# B&R Automation Studio project Snapshot
Automation Studio 4.9.2.46; technology packages: mapp 5.15.0, mappMotion 5.15.1

## Configuration Config1

CPU PC_any, AutomationRuntime D4.90, Build 4.1.2, Safety 0.0, Vc V4.72.2

### Task classes (Cpu.sw)
```
Cyclic#1 (cycle 10000 us):
  UserProgra <- UserProgram.prg
  TrakProgra <- TrakProgram.prg
  SV_Comms <- SV_Comms.prg
DataObjects: McAcpSys
Binaries: arsvcreg, udbdef, McAcpDrv, arflatprv, McProfGen, arcoal, FWRules, TCData, McAcpSim, ashwd, Config_1, ashwac, User, Config_4, sysconf, asfw, arconfig, iomap, Config_3, Config_2, Role, Config, Config_5
Libraries: McBase, McAxis, McAcpTrak, MpAxis, MpBase, McAcpAx, AsBrStr, TrakSnap, standard, MpRecipe, sys_lib, runtime, AsBrMath, powerlnk, astime, fileio, asepl, asieccon
```

### Hardware
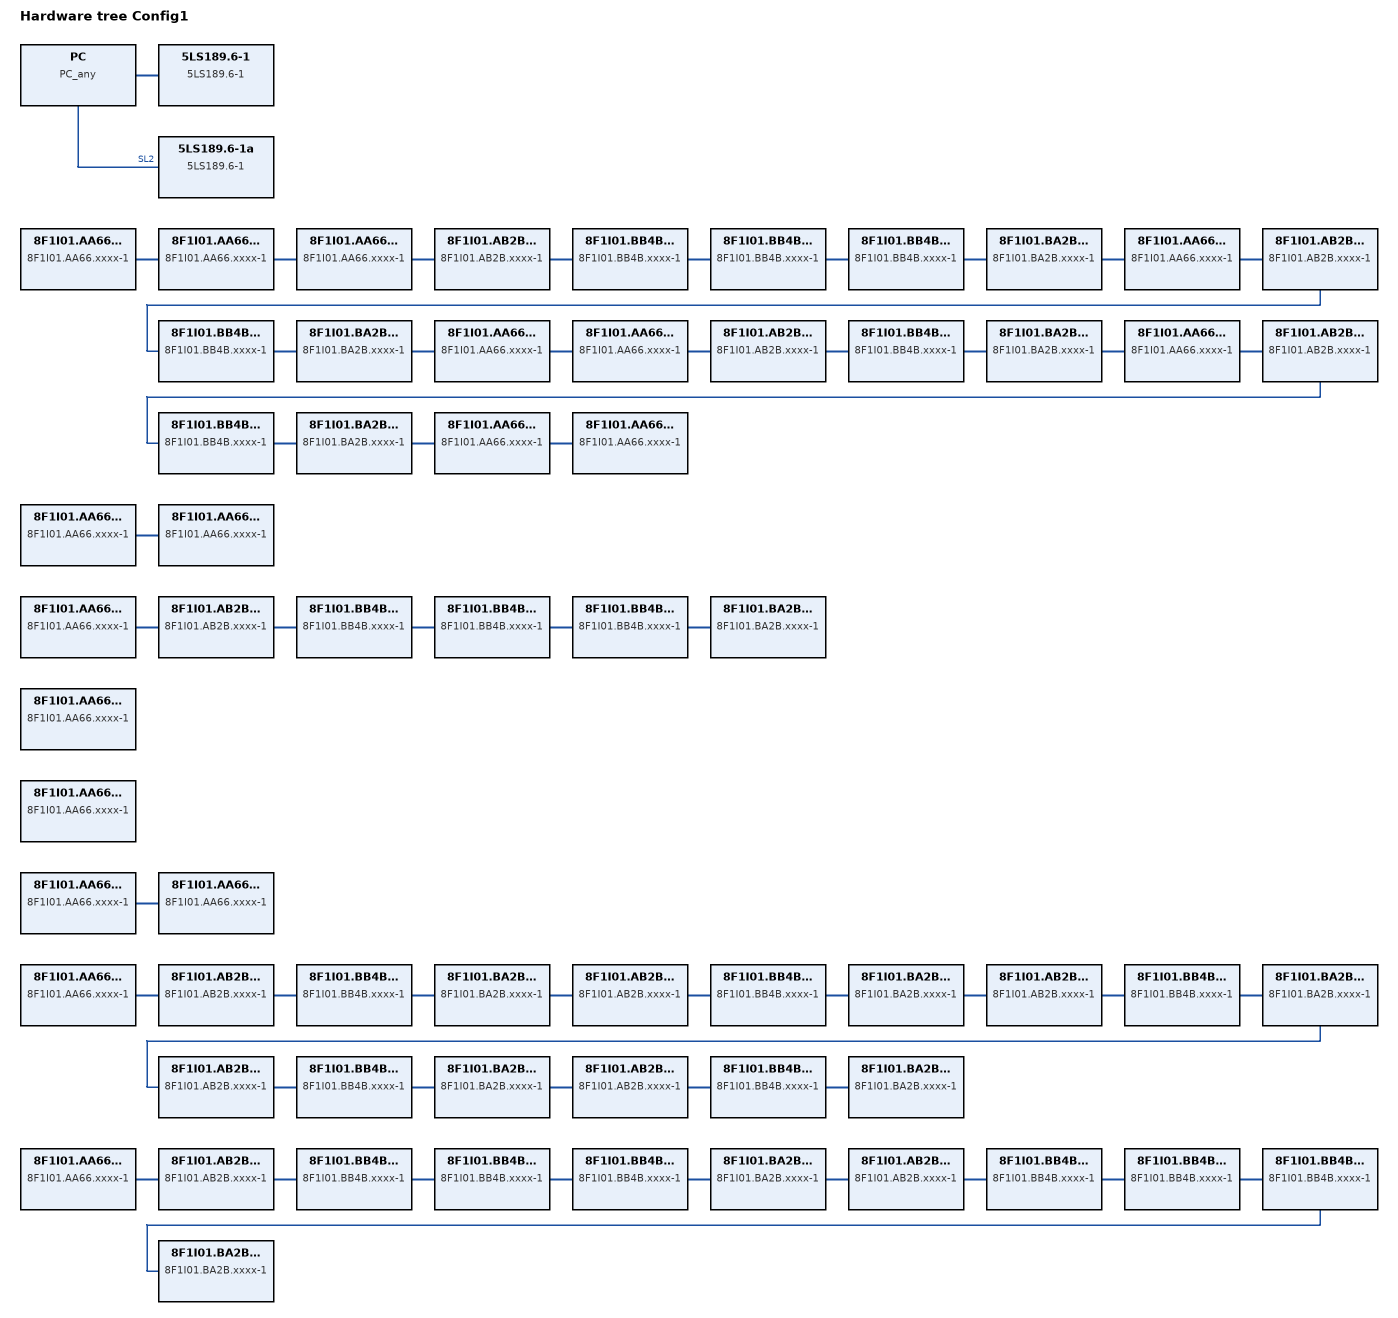
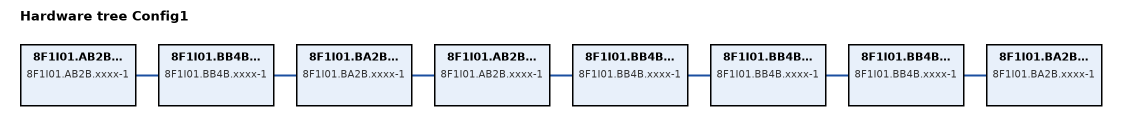
```
5LS189.6-1 : 5LS189.6-1 v1.4.1.0  [SL -> PC.SL1]
5LS189.6-1a : 5LS189.6-1 v1.4.1.0  [SL -> PC.SL2]
  Connector IF2:
    EplNatSubnet = 192.168.102.0
8F1I01.AA66.xxxx-1 : 8F1I01.AA66.xxxx-1 v1.0.0.2  [PLK1 -> 8F1I01.AA66.xxxx-1c.PLK2 [Cable Type=PowerlinkCable, Length=10, Version=1.0.0.3]; PLK2 -> 8F1I01.AA66.xxxx-1d.PLK1 [Cable Type=PowerlinkCable, Length=10, Version=1.0.0.3]]
  EnableDNA = on
  DriveConfiguration:
    McTypeID = LLMConfig
  DriveConfiguration/Segment:
    Shape = STRAIGHT660
    SegmentReference = SEG_13
    SegmentSectorReference = SECTOR_SEG_13
    SegmentSectorDirection = Positive
    ElongationCompensation = UseAssemblySetting
    StopReaction = UseAssemblySetting
    SpeedFilter = UseAssemblySetting
8F1I01.AA66.xxxx-1a : 8F1I01.AA66.xxxx-1 v1.0.0.2  [PLK1 -> 8F1I01.BA2B.xxxx-1a.PLK2 [Cable Type=PowerlinkCable, Length=10, Version=1.0.0.3]; PLK2 -> 8F1I01.AA66.xxxx-1c.PLK1 [Cable Type=PowerlinkCable, Length=10, Version=1.0.0.3]]
  EnableDNA = on
  DriveConfiguration:
    McTypeID = LLMConfig
  DriveConfiguration/Segment:
    Shape = STRAIGHT660
    SegmentReference = SEG_11
    SegmentSectorReference = SECTOR_SEG_11
    SegmentSectorDirection = Positive
    ElongationCompensation = UseAssemblySetting
    StopReaction = UseAssemblySetting
    SpeedFilter = UseAssemblySetting
8F1I01.AA66.xxxx-1b : 8F1I01.AA66.xxxx-1 v1.0.0.2  [PLK1 -> 8F1I01.AA66.xxxx-1d.PLK2 [Cable Type=PowerlinkCable, Length=10, Version=1.0.0.3]; PLK2 -> 8F1I01.AB2B.xxxx-1a.PLK1 [Cable Type=PowerlinkCable, Length=10, Version=1.0.0.3]]
  EnableDNA = on
  DriveConfiguration:
    McTypeID = LLMConfig
  DriveConfiguration/Segment:
    Shape = STRAIGHT660
    SegmentReference = SEG_15
    SegmentSectorReference = SECTOR_SEG_15
    SegmentSectorDirection = Positive
    ElongationCompensation = UseAssemblySetting
    StopReaction = UseAssemblySetting
    SpeedFilter = UseAssemblySetting
8F1I01.AA66.xxxx-1c : 8F1I01.AA66.xxxx-1 v1.0.0.2  [PLK1 -> 8F1I01.AA66.xxxx-1a.PLK2 [Cable Type=PowerlinkCable, Length=10, Version=1.0.0.3]; PLK2 -> 8F1I01.AA66.xxxx-1.PLK1 [Cable Type=PowerlinkCable, Length=10, Version=1.0.0.3]]
  EnableDNA = on
  DriveConfiguration:
    McTypeID = LLMConfig
  DriveConfiguration/Segment:
    Shape = STRAIGHT660
    SegmentReference = SEG_12
    SegmentSectorReference = SECTOR_SEG_12
    SegmentSectorDirection = Positive
    ElongationCompensation = UseAssemblySetting
    StopReaction = UseAssemblySetting
    SpeedFilter = UseAssemblySetting
8F1I01.AA66.xxxx-1d : 8F1I01.AA66.xxxx-1 v1.0.0.2  [PLK1 -> 8F1I01.AA66.xxxx-1.PLK2 [Cable Type=PowerlinkCable, Length=10, Version=1.0.0.3]; PLK2 -> 8F1I01.AA66.xxxx-1b.PLK1 [Cable Type=PowerlinkCable, Length=10, Version=1.0.0.3]]
  EnableDNA = on
  DriveConfiguration:
    McTypeID = LLMConfig
  DriveConfiguration/Segment:
    Shape = STRAIGHT660
    SegmentReference = SEG_14
    SegmentSectorReference = SECTOR_SEG_14
    SegmentSectorDirection = Positive
    ElongationCompensation = UseAssemblySetting
    StopReaction = UseAssemblySetting
    SpeedFilter = UseAssemblySetting
8F1I01.AA66.xxxx-1e : 8F1I01.AA66.xxxx-1 v1.0.0.2  [PLK1 -> 8F1I01.AA66.xxxx-1f.PLK2 [Cable Type=PowerlinkCable, Length=10, Version=1.0.0.3]; PLK2 -> 8F1I01.AB2B.xxxx-1.PLK1 [Cable Type=PowerlinkCable, Length=10, Version=1.0.0.3]]
  EnableDNA = on
  DriveConfiguration:
    McTypeID = LLMConfig
  DriveConfiguration/Segment:
    Shape = STRAIGHT660
    SegmentReference = SEG_05
    SegmentSectorReference = SECTOR_SEG_05
    SegmentSectorDirection = Positive
    ElongationCompensation = UseAssemblySetting
    StopReaction = UseAssemblySetting
    SpeedFilter = UseAssemblySetting
8F1I01.AA66.xxxx-1f : 8F1I01.AA66.xxxx-1 v1.0.0.2  [PLK1 -> 8F1I01.AA66.xxxx-1g.PLK2 [Cable Type=PowerlinkCable, Length=10, Version=1.0.0.3]; PLK2 -> 8F1I01.AA66.xxxx-1e.PLK1 [Cable Type=PowerlinkCable, Length=10, Version=1.0.0.3]]
  EnableDNA = on
  DriveConfiguration:
    McTypeID = LLMConfig
  DriveConfiguration/Segment:
    Shape = STRAIGHT660
    SegmentReference = SEG_04
    SegmentSectorReference = SECTOR_SEG_04
    SegmentSectorDirection = Positive
    ElongationCompensation = UseAssemblySetting
    StopReaction = UseAssemblySetting
    SpeedFilter = UseAssemblySetting
8F1I01.AA66.xxxx-1g : 8F1I01.AA66.xxxx-1 v1.0.0.2  [PLK1 -> 8F1I01.AA66.xxxx-1h.PLK2 [Cable Type=PowerlinkCable, Length=10, Version=1.0.0.3]; PLK2 -> 8F1I01.AA66.xxxx-1f.PLK1 [Cable Type=PowerlinkCable, Length=10, Version=1.0.0.3]]
  EnableDNA = on
  DriveConfiguration:
    McTypeID = LLMConfig
  DriveConfiguration/Segment:
    Shape = STRAIGHT660
    SegmentReference = SEG_03
    SegmentSectorReference = SECTOR_SEG_03
    SegmentSectorDirection = Positive
    ElongationCompensation = UseAssemblySetting
    StopReaction = UseAssemblySetting
    SpeedFilter = UseAssemblySetting
8F1I01.AA66.xxxx-1h : 8F1I01.AA66.xxxx-1 v1.0.0.2  [PLK1 -> 8F1I01.AA66.xxxx-1i.PLK2 [Cable Type=PowerlinkCable, Length=10, Version=1.0.0.3]; PLK2 -> 8F1I01.AA66.xxxx-1g.PLK1 [Cable Type=PowerlinkCable, Length=10, Version=1.0.0.3]]
  EnableDNA = on
  DriveConfiguration:
    McTypeID = LLMConfig
  DriveConfiguration/Segment:
    Shape = STRAIGHT660
    SegmentReference = SEG_02
    SegmentSectorReference = SECTOR_SEG_02
    SegmentSectorDirection = Positive
    ElongationCompensation = UseAssemblySetting
    StopReaction = UseAssemblySetting
    SpeedFilter = UseAssemblySetting
8F1I01.AA66.xxxx-1i : 8F1I01.AA66.xxxx-1 v1.0.0.2  [PLK2 -> 8F1I01.AA66.xxxx-1h.PLK1 [Cable Type=PowerlinkCable, Length=10, Version=1.0.0.3]; PLK3 -> 5LS189.6-1.IF2 [Cable Type=PowerlinkCable, Length=10, Version=1.0.0.3]]
  EnableDNA = on
  DriveConfiguration:
    McTypeID = LLMConfig
  DriveConfiguration/Segment:
    Shape = STRAIGHT660
    SegmentReference = SEG_01
    SegmentSectorReference = SECTOR_SEG_01
    SegmentSectorDirection = Positive
    ElongationCompensation = UseAssemblySetting
    StopReaction = UseAssemblySetting
    SpeedFilter = UseAssemblySetting
8F1I01.AA66.xxxx-1j : 8F1I01.AA66.xxxx-1 v1.0.0.2  [PLK1 -> 8F1I01.BA2B.xxxx-1.PLK2 [Cable Type=PowerlinkCable, Length=10, Version=1.0.0.3]; PLK2 -> 8F1I01.AB2B.xxxx-1b.PLK1 [Cable Type=PowerlinkCable, Length=10, Version=1.0.0.3]]
  EnableDNA = on
  DriveConfiguration:
    McTypeID = LLMConfig
  DriveConfiguration/Segment:
    Shape = STRAIGHT660
    SegmentReference = SEG_21
    SegmentSectorReference = SECTOR_SEG_21
    SegmentSectorDirection = Positive
    ElongationCompensation = UseAssemblySetting
    StopReaction = UseAssemblySetting
    SpeedFilter = UseAssemblySetting
8F1I01.AA66.xxxx-1k : 8F1I01.AA66.xxxx-1 v1.0.0.2  [PLK1 -> 8F1I01.AA66.xxxx-1l.PLK2 [Cable Type=PowerlinkCable, Length=10, Version=1.0.0.3]]
  EnableDNA = on
  DriveConfiguration:
    McTypeID = LLMConfig
  DriveConfiguration/Segment:
    Shape = STRAIGHT660
    SegmentReference = SEG_35
    SegmentSectorReference = SECTOR_SEG_35
    SegmentSectorDirection = Positive
    ElongationCompensation = UseAssemblySetting
    StopReaction = UseAssemblySetting
    SpeedFilter = UseAssemblySetting
8F1I01.AA66.xxxx-1l : 8F1I01.AA66.xxxx-1 v1.0.0.2  [PLK1 -> 8F1I01.BA2B.xxxx-1d.PLK2 [Cable Type=PowerlinkCable, Length=10, Version=1.0.0.3]; PLK2 -> 8F1I01.AA66.xxxx-1k.PLK1 [Cable Type=PowerlinkCable, Length=10, Version=1.0.0.3]]
  EnableDNA = on
  DriveConfiguration:
    McTypeID = LLMConfig
  DriveConfiguration/Segment:
    Shape = STRAIGHT660
    SegmentReference = SEG_34
    SegmentSectorReference = SECTOR_SEG_34
    SegmentSectorDirection = Positive
    ElongationCompensation = UseAssemblySetting
    StopReaction = UseAssemblySetting
    SpeedFilter = UseAssemblySetting
8F1I01.AA66.xxxx-1m : 8F1I01.AA66.xxxx-1 v1.0.0.2  [PLK1 -> 8F1I01.AA66.xxxx-1n.PLK2 [Cable Type=PowerlinkCable, Length=10, Version=1.0.0.3]; PLK2 -> 8F1I01.AB2B.xxxx-1d.PLK1 [Cable Type=PowerlinkCable, Length=10, Version=1.0.0.3]]
  EnableDNA = on
  DriveConfiguration:
    McTypeID = LLMConfig
  DriveConfiguration/Segment:
    Shape = STRAIGHT660
    SegmentReference = SEG_26
    SegmentSectorReference = SECTOR_SEG_26
    SegmentSectorDirection = Positive
    ElongationCompensation = UseAssemblySetting
    StopReaction = UseAssemblySetting
    SpeedFilter = UseAssemblySetting
8F1I01.AA66.xxxx-1n : 8F1I01.AA66.xxxx-1 v1.0.0.2  [PLK1 -> 8F1I01.BA2B.xxxx-1c.PLK2 [Cable Type=PowerlinkCable, Length=10, Version=1.0.0.3]; PLK2 -> 8F1I01.AA66.xxxx-1m.PLK1 [Cable Type=PowerlinkCable, Length=10, Version=1.0.0.3]]
  EnableDNA = on
  DriveConfiguration:
    McTypeID = LLMConfig
  DriveConfiguration/Segment:
    Shape = STRAIGHT660
    SegmentReference = SEG_25
    SegmentSectorReference = SECTOR_SEG_25
    SegmentSectorDirection = Positive
    ElongationCompensation = UseAssemblySetting
    StopReaction = UseAssemblySetting
    SpeedFilter = UseAssemblySetting
8F1I01.AA66.xxxx-1o : 8F1I01.AA66.xxxx-1 v1.0.0.2  [PLK1 -> 8F1I01.BA2B.xxxx-1e.PLK2 [Cable Type=PowerlinkCable, Length=10, Version=1.0.0.3]; PLK2 -> 8F1I01.AB2B.xxxx-1e.PLK1 [Cable Type=PowerlinkCable, Length=10, Version=1.0.0.3]]
  EnableDNA = on
  DriveConfiguration:
    McTypeID = LLMConfig
  DriveConfiguration/Segment:
    Shape = STRAIGHT660
    SegmentReference = SEG_30
    SegmentSectorReference = SECTOR_SEG_30
    SegmentSectorDirection = Positive
    ElongationCompensation = UseAssemblySetting
    StopReaction = UseAssemblySetting
    SpeedFilter = UseAssemblySetting
8F1I01.AA66.xxxx-1p : 8F1I01.AA66.xxxx-1 v1.0.0.2  [PLK1 -> 8F1I01.BA2B.xxxx-1f.PLK2 [Cable Type=PowerlinkCable, Length=10, Version=1.0.0.3]; PLK2 -> 8F1I01.AB2B.xxxx-1j.PLK1 [Cable Type=PowerlinkCable, Length=10, Version=1.0.0.3]]
  EnableDNA = on
  DriveConfiguration:
    McTypeID = LLMConfig
  DriveConfiguration/Segment:
    Shape = STRAIGHT660
    SegmentReference = SEG_55
    SegmentSectorReference = SECTOR_SEG_55
    SegmentSectorDirection = Positive
    ElongationCompensation = UseAssemblySetting
    StopReaction = UseAssemblySetting
    SpeedFilter = UseAssemblySetting
8F1I01.AA66.xxxx-1r : 8F1I01.AA66.xxxx-1 v1.0.0.2  [PLK1 -> 8F1I01.BA2B.xxxx-1k.PLK2 [Cable Type=PowerlinkCable, Length=10, Version=1.0.0.3]; PLK2 -> 8F1I01.AB2B.xxxx-1l.PLK1 [Cable Type=PowerlinkCable, Length=10, Version=1.0.0.3]]
  EnableDNA = on
  DriveConfiguration:
    McTypeID = LLMConfig
  DriveConfiguration/Segment:
    Shape = STRAIGHT660
    SegmentReference = SEG_44
    SegmentSectorReference = SECTOR_SEG_44
    SegmentSectorDirection = Positive
    ElongationCompensation = UseAssemblySetting
    StopReaction = UseAssemblySetting
    SpeedFilter = UseAssemblySetting
8F1I01.AB2B.xxxx-1 : 8F1I01.AB2B.xxxx-1 v1.0.0.2  [PLK1 -> 8F1I01.AA66.xxxx-1e.PLK2 [Cable Type=PowerlinkCable, Length=10, Version=1.0.0.3]; PLK2 -> 8F1I01.BB4B.xxxx-1b.PLK1 [Cable Type=PowerlinkCable, Length=10, Version=1.0.0.3]]
  EnableDNA = on
  DriveConfiguration:
    McTypeID = LLMConfig
  DriveConfiguration/Segment:
    Shape = STRAIGHT105_TO_CIRCULAR
    SegmentReference = SEG_06
    SegmentSectorReference = SECTOR_SEG_06
    SegmentSectorDirection = Positive
    ElongationCompensation = UseAssemblySetting
    StopReaction = UseAssemblySetting
    SpeedFilter = UseAssemblySetting
8F1I01.AB2B.xxxx-1a : 8F1I01.AB2B.xxxx-1 v1.0.0.2  [PLK1 -> 8F1I01.AA66.xxxx-1b.PLK2 [Cable Type=PowerlinkCable, Length=10, Version=1.0.0.3]; PLK2 -> 8F1I01.BB4B.xxxx-1e.PLK1 [Cable Type=PowerlinkCable, Length=10, Version=1.0.0.3]]
  EnableDNA = on
  DriveConfiguration:
    McTypeID = LLMConfig
  DriveConfiguration/Segment:
    Shape = STRAIGHT105_TO_CIRCULAR
    SegmentReference = SEG_16
    SegmentSectorReference = SECTOR_SEG_16
    SegmentSectorDirection = Positive
    ElongationCompensation = UseAssemblySetting
    StopReaction = UseAssemblySetting
    SpeedFilter = UseAssemblySetting
8F1I01.AB2B.xxxx-1b : 8F1I01.AB2B.xxxx-1 v1.0.0.2  [PLK1 -> 8F1I01.AA66.xxxx-1j.PLK2 [Cable Type=PowerlinkCable, Length=10, Version=1.0.0.3]; PLK2 -> 8F1I01.BB4B.xxxx-1f.PLK1 [Cable Type=PowerlinkCable, Length=10, Version=1.0.0.3]]
  EnableDNA = on
  DriveConfiguration:
    McTypeID = LLMConfig
  DriveConfiguration/Segment:
    Shape = STRAIGHT105_TO_CIRCULAR
    SegmentReference = SEG_22
    SegmentSectorReference = SECTOR_SEG_22
    SegmentSectorDirection = Positive
    ElongationCompensation = UseAssemblySetting
    StopReaction = UseAssemblySetting
    SpeedFilter = UseAssemblySetting
8F1I01.AB2B.xxxx-1c : 8F1I01.AB2B.xxxx-1 v1.0.0.2  [PLK2 -> 8F1I01.BB4B.xxxx-1g.PLK1 [Cable Type=PowerlinkCable, Length=10, Version=1.0.0.3]; PLK3 -> 5LS189.6-1a.IF2 [Cable Type=PowerlinkCable, Length=10, Version=1.0.0.3]]
  EnableDNA = on
  DriveConfiguration:
    McTypeID = LLMConfig
  DriveConfiguration/Segment:
    Shape = STRAIGHT105_TO_CIRCULAR
    SegmentReference = SEG_36
    SegmentSectorReference = SECTOR_SEG_36
    SegmentSectorDirection = Positive
    ElongationCompensation = UseAssemblySetting
    StopReaction = UseAssemblySetting
    SpeedFilter = UseAssemblySetting
8F1I01.AB2B.xxxx-1d : 8F1I01.AB2B.xxxx-1 v1.0.0.2  [PLK1 -> 8F1I01.AA66.xxxx-1m.PLK2 [Cable Type=PowerlinkCable, Length=10, Version=1.0.0.3]; PLK2 -> 8F1I01.BB4B.xxxx-1h.PLK1 [Cable Type=PowerlinkCable, Length=10, Version=1.0.0.3]]
  EnableDNA = on
  DriveConfiguration:
    McTypeID = LLMConfig
  DriveConfiguration/Segment:
    Shape = STRAIGHT105_TO_CIRCULAR
    SegmentReference = SEG_27
    SegmentSectorReference = SECTOR_SEG_27
    SegmentSectorDirection = Positive
    ElongationCompensation = UseAssemblySetting
    StopReaction = UseAssemblySetting
    SpeedFilter = UseAssemblySetting
8F1I01.AB2B.xxxx-1e : 8F1I01.AB2B.xxxx-1 v1.0.0.2  [PLK1 -> 8F1I01.AA66.xxxx-1o.PLK2 [Cable Type=PowerlinkCable, Length=10, Version=1.0.0.3]; PLK2 -> 8F1I01.BB4B.xxxx-1i.PLK1 [Cable Type=PowerlinkCable, Length=10, Version=1.0.0.3]]
  EnableDNA = on
  DriveConfiguration:
    McTypeID = LLMConfig
  DriveConfiguration/Segment:
    Shape = STRAIGHT105_TO_CIRCULAR
    SegmentReference = SEG_31
    SegmentSectorReference = SECTOR_SEG_31
    SegmentSectorDirection = Positive
    ElongationCompensation = UseAssemblySetting
    StopReaction = UseAssemblySetting
    SpeedFilter = UseAssemblySetting
8F1I01.AB2B.xxxx-1f : 8F1I01.AB2B.xxxx-1 v1.0.0.2  [PLK1 -> 8F1I01.BA2B.xxxx-1h.PLK2 [Cable Type=PowerlinkCable, Length=10, Version=1.0.0.3]; PLK2 -> 8F1I01.BB4B.xxxx-1l.PLK1 [Cable Type=PowerlinkCable, Length=10, Version=1.0.0.3]]
  EnableDNA = on
  DriveConfiguration:
    McTypeID = LLMConfig
  DriveConfiguration/Segment:
    Shape = STRAIGHT105_TO_CIRCULAR
    SegmentReference = SEG_68
    SegmentSectorReference = SECTOR_SEG_68
    SegmentSectorDirection = Positive
    ElongationCompensation = UseAssemblySetting
    StopReaction = UseAssemblySetting
    SpeedFilter = UseAssemblySetting
8F1I01.AB2B.xxxx-1g : 8F1I01.AB2B.xxxx-1 v1.0.0.2  [PLK1 -> 8F1I01.BA2B.xxxx-1j.PLK2 [Cable Type=PowerlinkCable, Length=10, Version=1.0.0.3]; PLK2 -> 8F1I01.BB4B.xxxx-1k.PLK1 [Cable Type=PowerlinkCable, Length=10, Version=1.0.0.3]]
  EnableDNA = on
  DriveConfiguration:
    McTypeID = LLMConfig
  DriveConfiguration/Segment:
    Shape = STRAIGHT105_TO_CIRCULAR
    SegmentReference = SEG_62
    SegmentSectorReference = SECTOR_SEG_62
    SegmentSectorDirection = Positive
    ElongationCompensation = UseAssemblySetting
    StopReaction = UseAssemblySetting
    SpeedFilter = UseAssemblySetting
8F1I01.AB2B.xxxx-1h : 8F1I01.AB2B.xxxx-1 v1.0.0.2  [PLK1 -> 8F1I01.BA2B.xxxx-1g.PLK2 [Cable Type=PowerlinkCable, Length=10, Version=1.0.0.3]; PLK2 -> 8F1I01.BB4B.xxxx-1x.PLK1 [Cable Type=PowerlinkCable, Length=10, Version=1.0.0.3]]
  EnableDNA = on
  DriveConfiguration:
    McTypeID = LLMConfig
  DriveConfiguration/Segment:
    Shape = STRAIGHT105_TO_CIRCULAR
    SegmentReference = SEG_65
    SegmentSectorReference = SECTOR_SEG_65
    SegmentSectorDirection = Positive
    ElongationCompensation = UseAssemblySetting
    StopReaction = UseAssemblySetting
    SpeedFilter = UseAssemblySetting
8F1I01.AB2B.xxxx-1i : 8F1I01.AB2B.xxxx-1 v1.0.0.2  [PLK1 -> 8F1I01.BA2B.xxxx-1i.PLK2 [Cable Type=PowerlinkCable, Length=10, Version=1.0.0.3]; PLK2 -> 8F1I01.BB4B.xxxx-1n.PLK1 [Cable Type=PowerlinkCable, Length=10, Version=1.0.0.3]]
  EnableDNA = on
  DriveConfiguration:
    McTypeID = LLMConfig
  DriveConfiguration/Segment:
    Shape = STRAIGHT105_TO_CIRCULAR
    SegmentReference = SEG_59
    SegmentSectorReference = SECTOR_SEG_59
    SegmentSectorDirection = Positive
    ElongationCompensation = UseAssemblySetting
    StopReaction = UseAssemblySetting
    SpeedFilter = UseAssemblySetting
8F1I01.AB2B.xxxx-1j : 8F1I01.AB2B.xxxx-1 v1.0.0.2  [PLK1 -> 8F1I01.AA66.xxxx-1p.PLK2 [Cable Type=PowerlinkCable, Length=10, Version=1.0.0.3]; PLK2 -> 8F1I01.BB4B.xxxx-1m.PLK1 [Cable Type=PowerlinkCable, Length=10, Version=1.0.0.3]]
  EnableDNA = on
  DriveConfiguration:
    McTypeID = LLMConfig
  DriveConfiguration/Segment:
    Shape = STRAIGHT105_TO_CIRCULAR
    SegmentReference = SEG_56
    SegmentSectorReference = SECTOR_SEG_56
    SegmentSectorDirection = Positive
    ElongationCompensation = UseAssemblySetting
    StopReaction = UseAssemblySetting
    SpeedFilter = UseAssemblySetting
8F1I01.AB2B.xxxx-1k : 8F1I01.AB2B.xxxx-1 v1.0.0.2  [PLK1 -> 8F1I01.BA2B.xxxx-1b.PLK2 [Cable Type=PowerlinkCable, Length=10, Version=1.0.0.3]; PLK2 -> 8F1I01.BB4B.xxxx-1o.PLK1 [Cable Type=PowerlinkCable, Length=10, Version=1.0.0.3]]
  EnableDNA = on
  DriveConfiguration:
    McTypeID = LLMConfig
  DriveConfiguration/Segment:
    Shape = STRAIGHT105_TO_CIRCULAR
    SegmentReference = SEG_39
    SegmentSectorReference = SECTOR_SEG_39
    SegmentSectorDirection = Positive
    ElongationCompensation = UseAssemblySetting
    StopReaction = UseAssemblySetting
    SpeedFilter = UseAssemblySetting
8F1I01.AB2B.xxxx-1l : 8F1I01.AB2B.xxxx-1 v1.0.0.2  [PLK1 -> 8F1I01.AA66.xxxx-1r.PLK2 [Cable Type=PowerlinkCable, Length=10, Version=1.0.0.3]; PLK2 -> 8F1I01.BB4B.xxxx-1r.PLK1 [Cable Type=PowerlinkCable, Length=10, Version=1.0.0.3]]
  EnableDNA = on
  DriveConfiguration:
    McTypeID = LLMConfig
  DriveConfiguration/Segment:
    Shape = STRAIGHT105_TO_CIRCULAR
    SegmentReference = SEG_45
    SegmentSectorReference = SECTOR_SEG_45
    SegmentSectorDirection = Positive
    ElongationCompensation = UseAssemblySetting
    StopReaction = UseAssemblySetting
    SpeedFilter = UseAssemblySetting
8F1I01.AB2B.xxxx-1m : 8F1I01.AB2B.xxxx-1 v1.0.0.2  [PLK1 -> 8F1I01.BA2B.xxxx-1l.PLK2 [Cable Type=PowerlinkCable, Length=10, Version=1.0.0.3]; PLK2 -> 8F1I01.BB4B.xxxx-1v.PLK1 [Cable Type=PowerlinkCable, Length=10, Version=1.0.0.3]]
  EnableDNA = on
  DriveConfiguration:
    McTypeID = LLMConfig
  DriveConfiguration/Segment:
    Shape = STRAIGHT105_TO_CIRCULAR
    SegmentReference = SEG_50
    SegmentSectorReference = SECTOR_SEG_50
    SegmentSectorDirection = Positive
    ElongationCompensation = UseAssemblySetting
    StopReaction = UseAssemblySetting
    SpeedFilter = UseAssemblySetting
8F1I01.BA2B.xxxx-1 : 8F1I01.BA2B.xxxx-1 v1.0.0.2  [PLK1 -> 8F1I01.BB4B.xxxx-1c.PLK2 [Cable Type=PowerlinkCable, Length=10, Version=1.0.0.3]; PLK2 -> 8F1I01.AA66.xxxx-1j.PLK1 [Cable Type=PowerlinkCable, Length=10, Version=1.0.0.3]]
  EnableDNA = on
  DriveConfiguration:
    McTypeID = LLMConfig
  DriveConfiguration/Segment:
    Shape = CIRCULAR_TO_STRAIGHT105
    SegmentReference = SEG_20
    SegmentSectorReference = SECTOR_SEG_20
    SegmentSectorDirection = Positive
    ElongationCompensation = UseAssemblySetting
    StopReaction = UseAssemblySetting
    SpeedFilter = UseAssemblySetting
8F1I01.BA2B.xxxx-1a : 8F1I01.BA2B.xxxx-1 v1.0.0.2  [PLK1 -> 8F1I01.BB4B.xxxx-1.PLK2 [Cable Type=PowerlinkCable, Length=10, Version=1.0.0.3]; PLK2 -> 8F1I01.AA66.xxxx-1a.PLK1 [Cable Type=PowerlinkCable, Length=10, Version=1.0.0.3]]
  EnableDNA = on
  DriveConfiguration:
    McTypeID = LLMConfig
  DriveConfiguration/Segment:
    Shape = CIRCULAR_TO_STRAIGHT105
    SegmentReference = SEG_10
    SegmentSectorReference = SECTOR_SEG_10
    SegmentSectorDirection = Positive
    ElongationCompensation = UseAssemblySetting
    StopReaction = UseAssemblySetting
    SpeedFilter = UseAssemblySetting
8F1I01.BA2B.xxxx-1b : 8F1I01.BA2B.xxxx-1 v1.0.0.2  [PLK1 -> 8F1I01.BB4B.xxxx-1g.PLK2 [Cable Type=PowerlinkCable, Length=10, Version=1.0.0.3]; PLK2 -> 8F1I01.AB2B.xxxx-1k.PLK1 [Cable Type=PowerlinkCable, Length=10, Version=1.0.0.3]]
  EnableDNA = on
  DriveConfiguration:
    McTypeID = LLMConfig
  DriveConfiguration/Segment:
    Shape = CIRCULAR_TO_STRAIGHT105
    SegmentReference = SEG_38
    SegmentSectorReference = SECTOR_SEG_38
    SegmentSectorDirection = Positive
    ElongationCompensation = UseAssemblySetting
    StopReaction = UseAssemblySetting
    SpeedFilter = UseAssemblySetting
8F1I01.BA2B.xxxx-1c : 8F1I01.BA2B.xxxx-1 v1.0.0.2  [PLK1 -> 8F1I01.BB4B.xxxx-1f.PLK2 [Cable Type=PowerlinkCable, Length=10, Version=1.0.0.3]; PLK2 -> 8F1I01.AA66.xxxx-1n.PLK1 [Cable Type=PowerlinkCable, Length=10, Version=1.0.0.3]]
  EnableDNA = on
  DriveConfiguration:
    McTypeID = LLMConfig
  DriveConfiguration/Segment:
    Shape = CIRCULAR_TO_STRAIGHT105
    SegmentReference = SEG_24
    SegmentSectorReference = SECTOR_SEG_24
    SegmentSectorDirection = Positive
    ElongationCompensation = UseAssemblySetting
    StopReaction = UseAssemblySetting
    SpeedFilter = UseAssemblySetting
8F1I01.BA2B.xxxx-1d : 8F1I01.BA2B.xxxx-1 v1.0.0.2  [PLK1 -> 8F1I01.BB4B.xxxx-1i.PLK2 [Cable Type=PowerlinkCable, Length=10, Version=1.0.0.3]; PLK2 -> 8F1I01.AA66.xxxx-1l.PLK1 [Cable Type=PowerlinkCable, Length=10, Version=1.0.0.3]]
  EnableDNA = on
  DriveConfiguration:
    McTypeID = LLMConfig
  DriveConfiguration/Segment:
    Shape = CIRCULAR_TO_STRAIGHT105
    SegmentReference = SEG_33
    SegmentSectorReference = SECTOR_SEG_33
    SegmentSectorDirection = Positive
    ElongationCompensation = UseAssemblySetting
    StopReaction = UseAssemblySetting
    SpeedFilter = UseAssemblySetting
8F1I01.BA2B.xxxx-1e : 8F1I01.BA2B.xxxx-1 v1.0.0.2  [PLK1 -> 8F1I01.BB4B.xxxx-1h.PLK2 [Cable Type=PowerlinkCable, Length=10, Version=1.0.0.3]; PLK2 -> 8F1I01.AA66.xxxx-1o.PLK1 [Cable Type=PowerlinkCable, Length=10, Version=1.0.0.3]]
  EnableDNA = on
  DriveConfiguration:
    McTypeID = LLMConfig
  DriveConfiguration/Segment:
    Shape = CIRCULAR_TO_STRAIGHT105
    SegmentReference = SEG_29
    SegmentSectorReference = SECTOR_SEG_29
    SegmentSectorDirection = Positive
    ElongationCompensation = UseAssemblySetting
    StopReaction = UseAssemblySetting
    SpeedFilter = UseAssemblySetting
8F1I01.BA2B.xxxx-1f : 8F1I01.BA2B.xxxx-1 v1.0.0.2  [PLK1 -> 8F1I01.BB4B.xxxx-1u.PLK2 [Cable Type=PowerlinkCable, Length=10, Version=1.0.0.3]; PLK2 -> 8F1I01.AA66.xxxx-1p.PLK1 [Cable Type=PowerlinkCable, Length=10, Version=1.0.0.3]]
  EnableDNA = on
  DriveConfiguration:
    McTypeID = LLMConfig
  DriveConfiguration/Segment:
    Shape = CIRCULAR_TO_STRAIGHT105
    SegmentReference = SEG_54
    SegmentSectorReference = SECTOR_SEG_54
    SegmentSectorDirection = Positive
    ElongationCompensation = UseAssemblySetting
    StopReaction = UseAssemblySetting
    SpeedFilter = UseAssemblySetting
8F1I01.BA2B.xxxx-1g : 8F1I01.BA2B.xxxx-1 v1.0.0.2  [PLK1 -> 8F1I01.BB4B.xxxx-1k.PLK2 [Cable Type=PowerlinkCable, Length=10, Version=1.0.0.3]; PLK2 -> 8F1I01.AB2B.xxxx-1h.PLK1 [Cable Type=PowerlinkCable, Length=10, Version=1.0.0.3]]
  EnableDNA = on
  DriveConfiguration:
    McTypeID = LLMConfig
  DriveConfiguration/Segment:
    Shape = CIRCULAR_TO_STRAIGHT105
    SegmentReference = SEG_64
    SegmentSectorReference = SECTOR_SEG_64
    SegmentSectorDirection = Positive
    ElongationCompensation = UseAssemblySetting
    StopReaction = UseAssemblySetting
    SpeedFilter = UseAssemblySetting
8F1I01.BA2B.xxxx-1h : 8F1I01.BA2B.xxxx-1 v1.0.0.2  [PLK1 -> 8F1I01.BB4B.xxxx-1x.PLK2 [Cable Type=PowerlinkCable, Length=10, Version=1.0.0.3]; PLK2 -> 8F1I01.AB2B.xxxx-1f.PLK1 [Cable Type=PowerlinkCable, Length=10, Version=1.0.0.3]]
  EnableDNA = on
  DriveConfiguration:
    McTypeID = LLMConfig
  DriveConfiguration/Segment:
    Shape = CIRCULAR_TO_STRAIGHT105
    SegmentReference = SEG_67
    SegmentSectorReference = SECTOR_SEG_67
    SegmentSectorDirection = Positive
    ElongationCompensation = UseAssemblySetting
    StopReaction = UseAssemblySetting
    SpeedFilter = UseAssemblySetting
8F1I01.BA2B.xxxx-1i : 8F1I01.BA2B.xxxx-1 v1.0.0.2  [PLK1 -> 8F1I01.BB4B.xxxx-1m.PLK2 [Cable Type=PowerlinkCable, Length=10, Version=1.0.0.3]; PLK2 -> 8F1I01.AB2B.xxxx-1i.PLK1 [Cable Type=PowerlinkCable, Length=10, Version=1.0.0.3]]
  EnableDNA = on
  DriveConfiguration:
    McTypeID = LLMConfig
  DriveConfiguration/Segment:
    Shape = CIRCULAR_TO_STRAIGHT105
    SegmentReference = SEG_58
    SegmentSectorReference = SECTOR_SEG_58
    SegmentSectorDirection = Positive
    ElongationCompensation = UseAssemblySetting
    StopReaction = UseAssemblySetting
    SpeedFilter = UseAssemblySetting
8F1I01.BA2B.xxxx-1j : 8F1I01.BA2B.xxxx-1 v1.0.0.2  [PLK1 -> 8F1I01.BB4B.xxxx-1n.PLK2 [Cable Type=PowerlinkCable, Length=10, Version=1.0.0.3]; PLK2 -> 8F1I01.AB2B.xxxx-1g.PLK1 [Cable Type=PowerlinkCable, Length=10, Version=1.0.0.3]]
  EnableDNA = on
  DriveConfiguration:
    McTypeID = LLMConfig
  DriveConfiguration/Segment:
    Shape = CIRCULAR_TO_STRAIGHT105
    SegmentReference = SEG_61
    SegmentSectorReference = SECTOR_SEG_61
    SegmentSectorDirection = Positive
    ElongationCompensation = UseAssemblySetting
    StopReaction = UseAssemblySetting
    SpeedFilter = UseAssemblySetting
8F1I01.BA2B.xxxx-1k : 8F1I01.BA2B.xxxx-1 v1.0.0.2  [PLK1 -> 8F1I01.BB4B.xxxx-1s.PLK2 [Cable Type=PowerlinkCable, Length=10, Version=1.0.0.3]; PLK2 -> 8F1I01.AA66.xxxx-1r.PLK1 [Cable Type=PowerlinkCable, Length=10, Version=1.0.0.3]]
  EnableDNA = on
  DriveConfiguration:
    McTypeID = LLMConfig
  DriveConfiguration/Segment:
    Shape = CIRCULAR_TO_STRAIGHT105
    SegmentReference = SEG_43
    SegmentSectorReference = SECTOR_SEG_43
    SegmentSectorDirection = Positive
    ElongationCompensation = UseAssemblySetting
    StopReaction = UseAssemblySetting
    SpeedFilter = UseAssemblySetting
8F1I01.BA2B.xxxx-1l : 8F1I01.BA2B.xxxx-1 v1.0.0.2  [PLK1 -> 8F1I01.BB4B.xxxx-1p.PLK2 [Cable Type=PowerlinkCable, Length=10, Version=1.0.0.3]; PLK2 -> 8F1I01.AB2B.xxxx-1m.PLK1 [Cable Type=PowerlinkCable, Length=10, Version=1.0.0.3]]
  EnableDNA = on
  DriveConfiguration:
    McTypeID = LLMConfig
  DriveConfiguration/Segment:
    Shape = CIRCULAR_TO_STRAIGHT105
    SegmentReference = SEG_49
    SegmentSectorReference = SECTOR_SEG_49
    SegmentSectorDirection = Positive
    ElongationCompensation = UseAssemblySetting
    StopReaction = UseAssemblySetting
    SpeedFilter = UseAssemblySetting
8F1I01.BA2B.xxxx-1m : 8F1I01.BA2B.xxxx-1 v1.0.0.2  [PLK1 -> 8F1I01.BB4B.xxxx-1l.PLK2 [Cable Type=PowerlinkCable, Length=10, Version=1.0.0.3]]
  EnableDNA = on
  DriveConfiguration:
    McTypeID = LLMConfig
  DriveConfiguration/Segment:
    Shape = CIRCULAR_TO_STRAIGHT105
    SegmentReference = SEG_70
    SegmentSectorReference = SECTOR_SEG_70
    SegmentSectorDirection = Positive
    ElongationCompensation = UseAssemblySetting
    StopReaction = UseAssemblySetting
    SpeedFilter = UseAssemblySetting
8F1I01.BB4B.xxxx-1 : 8F1I01.BB4B.xxxx-1 v1.0.0.2  [PLK1 -> 8F1I01.BB4B.xxxx-1a.PLK2 [Cable Type=PowerlinkCable, Length=10, Version=1.0.0.3]; PLK2 -> 8F1I01.BA2B.xxxx-1a.PLK1 [Cable Type=PowerlinkCable, Length=10, Version=1.0.0.3]]
  EnableDNA = on
  DriveConfiguration:
    McTypeID = LLMConfig
  DriveConfiguration/Segment:
    Shape = CIRCULAR
    SegmentReference = SEG_09
    SegmentSectorReference = SECTOR_SEG_09
    SegmentSectorDirection = Positive
    ElongationCompensation = UseAssemblySetting
    StopReaction = UseAssemblySetting
    SpeedFilter = UseAssemblySetting
8F1I01.BB4B.xxxx-1a : 8F1I01.BB4B.xxxx-1 v1.0.0.2  [PLK1 -> 8F1I01.BB4B.xxxx-1b.PLK2 [Cable Type=PowerlinkCable, Length=10, Version=1.0.0.3]; PLK2 -> 8F1I01.BB4B.xxxx-1.PLK1 [Cable Type=PowerlinkCable, Length=10, Version=1.0.0.3]]
  EnableDNA = on
  DriveConfiguration:
    McTypeID = LLMConfig
  DriveConfiguration/Segment:
    Shape = CIRCULAR
    SegmentReference = SEG_08
    SegmentSectorReference = SECTOR_SEG_08
    SegmentSectorDirection = Positive
    ElongationCompensation = UseAssemblySetting
    StopReaction = UseAssemblySetting
    SpeedFilter = UseAssemblySetting
8F1I01.BB4B.xxxx-1b : 8F1I01.BB4B.xxxx-1 v1.0.0.2  [PLK1 -> 8F1I01.AB2B.xxxx-1.PLK2 [Cable Type=PowerlinkCable, Length=10, Version=1.0.0.3]; PLK2 -> 8F1I01.BB4B.xxxx-1a.PLK1 [Cable Type=PowerlinkCable, Length=10, Version=1.0.0.3]]
  EnableDNA = on
  DriveConfiguration:
    McTypeID = LLMConfig
  DriveConfiguration/Segment:
    Shape = CIRCULAR
    SegmentReference = SEG_07
    SegmentSectorReference = SECTOR_SEG_07
    SegmentSectorDirection = Positive
    ElongationCompensation = UseAssemblySetting
    StopReaction = UseAssemblySetting
    SpeedFilter = UseAssemblySetting
8F1I01.BB4B.xxxx-1c : 8F1I01.BB4B.xxxx-1 v1.0.0.2  [PLK1 -> 8F1I01.BB4B.xxxx-1d.PLK2 [Cable Type=PowerlinkCable, Length=10, Version=1.0.0.3]; PLK2 -> 8F1I01.BA2B.xxxx-1.PLK1 [Cable Type=PowerlinkCable, Length=10, Version=1.0.0.3]]
  EnableDNA = on
  DriveConfiguration:
    McTypeID = LLMConfig
  DriveConfiguration/Segment:
    Shape = CIRCULAR
    SegmentReference = SEG_19
    SegmentSectorReference = SECTOR_SEG_19
    SegmentSectorDirection = Positive
    ElongationCompensation = UseAssemblySetting
    StopReaction = UseAssemblySetting
    SpeedFilter = UseAssemblySetting
8F1I01.BB4B.xxxx-1d : 8F1I01.BB4B.xxxx-1 v1.0.0.2  [PLK1 -> 8F1I01.BB4B.xxxx-1e.PLK2 [Cable Type=PowerlinkCable, Length=10, Version=1.0.0.3]; PLK2 -> 8F1I01.BB4B.xxxx-1c.PLK1 [Cable Type=PowerlinkCable, Length=10, Version=1.0.0.3]]
  EnableDNA = on
  DriveConfiguration:
    McTypeID = LLMConfig
  DriveConfiguration/Segment:
    Shape = CIRCULAR
    SegmentReference = SEG_18
    SegmentSectorReference = SECTOR_SEG_18
    SegmentSectorDirection = Positive
    ElongationCompensation = UseAssemblySetting
    StopReaction = UseAssemblySetting
    SpeedFilter = UseAssemblySetting
8F1I01.BB4B.xxxx-1e : 8F1I01.BB4B.xxxx-1 v1.0.0.2  [PLK1 -> 8F1I01.AB2B.xxxx-1a.PLK2 [Cable Type=PowerlinkCable, Length=10, Version=1.0.0.3]; PLK2 -> 8F1I01.BB4B.xxxx-1d.PLK1 [Cable Type=PowerlinkCable, Length=10, Version=1.0.0.3]]
  EnableDNA = on
  DriveConfiguration:
    McTypeID = LLMConfig
  DriveConfiguration/Segment:
    Shape = CIRCULAR
    SegmentReference = SEG_17
    SegmentSectorReference = SECTOR_SEG_17
    SegmentSectorDirection = Positive
    ElongationCompensation = UseAssemblySetting
    StopReaction = UseAssemblySetting
    SpeedFilter = UseAssemblySetting
8F1I01.BB4B.xxxx-1f : 8F1I01.BB4B.xxxx-1 v1.0.0.2  [PLK1 -> 8F1I01.AB2B.xxxx-1b.PLK2 [Cable Type=PowerlinkCable, Length=10, Version=1.0.0.3]; PLK2 -> 8F1I01.BA2B.xxxx-1c.PLK1 [Cable Type=PowerlinkCable, Length=10, Version=1.0.0.3]]
  EnableDNA = on
  DriveConfiguration:
    McTypeID = LLMConfig
  DriveConfiguration/Segment:
    Shape = CIRCULAR
    SegmentReference = SEG_23
    SegmentSectorReference = SECTOR_SEG_23
    SegmentSectorDirection = Positive
    ElongationCompensation = UseAssemblySetting
    StopReaction = UseAssemblySetting
    SpeedFilter = UseAssemblySetting
8F1I01.BB4B.xxxx-1g : 8F1I01.BB4B.xxxx-1 v1.0.0.2  [PLK1 -> 8F1I01.AB2B.xxxx-1c.PLK2 [Cable Type=PowerlinkCable, Length=10, Version=1.0.0.3]; PLK2 -> 8F1I01.BA2B.xxxx-1b.PLK1 [Cable Type=PowerlinkCable, Length=10, Version=1.0.0.3]]
  EnableDNA = on
  DriveConfiguration:
    McTypeID = LLMConfig
  DriveConfiguration/Segment:
    Shape = CIRCULAR
    SegmentReference = SEG_37
    SegmentSectorReference = SECTOR_SEG_37
    SegmentSectorDirection = Positive
    ElongationCompensation = UseAssemblySetting
    StopReaction = UseAssemblySetting
    SpeedFilter = UseAssemblySetting
8F1I01.BB4B.xxxx-1h : 8F1I01.BB4B.xxxx-1 v1.0.0.2  [PLK1 -> 8F1I01.AB2B.xxxx-1d.PLK2 [Cable Type=PowerlinkCable, Length=10, Version=1.0.0.3]; PLK2 -> 8F1I01.BA2B.xxxx-1e.PLK1 [Cable Type=PowerlinkCable, Length=10, Version=1.0.0.3]]
  EnableDNA = on
  DriveConfiguration:
    McTypeID = LLMConfig
  DriveConfiguration/Segment:
    Shape = CIRCULAR
    SegmentReference = SEG_28
    SegmentSectorReference = SECTOR_SEG_28
    SegmentSectorDirection = Positive
    ElongationCompensation = UseAssemblySetting
    StopReaction = UseAssemblySetting
    SpeedFilter = UseAssemblySetting
8F1I01.BB4B.xxxx-1i : 8F1I01.BB4B.xxxx-1 v1.0.0.2  [PLK1 -> 8F1I01.AB2B.xxxx-1e.PLK2 [Cable Type=PowerlinkCable, Length=10, Version=1.0.0.3]; PLK2 -> 8F1I01.BA2B.xxxx-1d.PLK1 [Cable Type=PowerlinkCable, Length=10, Version=1.0.0.3]]
  EnableDNA = on
  DriveConfiguration:
    McTypeID = LLMConfig
  DriveConfiguration/Segment:
    Shape = CIRCULAR
    SegmentReference = SEG_32
    SegmentSectorReference = SECTOR_SEG_32
    SegmentSectorDirection = Positive
    ElongationCompensation = UseAssemblySetting
    StopReaction = UseAssemblySetting
    SpeedFilter = UseAssemblySetting
8F1I01.BB4B.xxxx-1j : 8F1I01.BB4B.xxxx-1 v1.0.0.2  [PLK1 -> 8F1I01.BB4B.xxxx-1v.PLK2 [Cable Type=PowerlinkCable, Length=10, Version=1.0.0.3]; PLK2 -> 8F1I01.BB4B.xxxx-1u.PLK1 [Cable Type=PowerlinkCable, Length=10, Version=1.0.0.3]]
  EnableDNA = on
  DriveConfiguration:
    McTypeID = LLMConfig
  DriveConfiguration/Segment:
    Shape = CIRCULAR
    SegmentReference = SEG_52
    SegmentSectorReference = SECTOR_SEG_52
    SegmentSectorDirection = Positive
    ElongationCompensation = UseAssemblySetting
    StopReaction = UseAssemblySetting
    SpeedFilter = UseAssemblySetting
8F1I01.BB4B.xxxx-1k : 8F1I01.BB4B.xxxx-1 v1.0.0.2  [PLK1 -> 8F1I01.AB2B.xxxx-1g.PLK2 [Cable Type=PowerlinkCable, Length=10, Version=1.0.0.3]; PLK2 -> 8F1I01.BA2B.xxxx-1g.PLK1 [Cable Type=PowerlinkCable, Length=10, Version=1.0.0.3]]
  EnableDNA = on
  DriveConfiguration:
    McTypeID = LLMConfig
  DriveConfiguration/Segment:
    Shape = CIRCULAR
    SegmentReference = SEG_63
    SegmentSectorReference = SECTOR_SEG_63
    SegmentSectorDirection = Positive
    ElongationCompensation = UseAssemblySetting
    StopReaction = UseAssemblySetting
    SpeedFilter = UseAssemblySetting
8F1I01.BB4B.xxxx-1l : 8F1I01.BB4B.xxxx-1 v1.0.0.2  [PLK1 -> 8F1I01.AB2B.xxxx-1f.PLK2 [Cable Type=PowerlinkCable, Length=10, Version=1.0.0.3]; PLK2 -> 8F1I01.BA2B.xxxx-1m.PLK1 [Cable Type=PowerlinkCable, Length=10, Version=1.0.0.3]]
  EnableDNA = on
  DriveConfiguration:
    McTypeID = LLMConfig
  DriveConfiguration/Segment:
    Shape = CIRCULAR
    SegmentReference = SEG_69
    SegmentSectorReference = SECTOR_SEG_69
    SegmentSectorDirection = Positive
    ElongationCompensation = UseAssemblySetting
    StopReaction = UseAssemblySetting
    SpeedFilter = UseAssemblySetting
8F1I01.BB4B.xxxx-1m : 8F1I01.BB4B.xxxx-1 v1.0.0.2  [PLK1 -> 8F1I01.AB2B.xxxx-1j.PLK2 [Cable Type=PowerlinkCable, Length=10, Version=1.0.0.3]; PLK2 -> 8F1I01.BA2B.xxxx-1i.PLK1 [Cable Type=PowerlinkCable, Length=10, Version=1.0.0.3]]
  EnableDNA = on
  DriveConfiguration:
    McTypeID = LLMConfig
  DriveConfiguration/Segment:
    Shape = CIRCULAR
    SegmentReference = SEG_57
    SegmentSectorReference = SECTOR_SEG_57
    SegmentSectorDirection = Positive
    ElongationCompensation = UseAssemblySetting
    StopReaction = UseAssemblySetting
    SpeedFilter = UseAssemblySetting
8F1I01.BB4B.xxxx-1n : 8F1I01.BB4B.xxxx-1 v1.0.0.2  [PLK1 -> 8F1I01.AB2B.xxxx-1i.PLK2 [Cable Type=PowerlinkCable, Length=10, Version=1.0.0.3]; PLK2 -> 8F1I01.BA2B.xxxx-1j.PLK1 [Cable Type=PowerlinkCable, Length=10, Version=1.0.0.3]]
  EnableDNA = on
  DriveConfiguration:
    McTypeID = LLMConfig
  DriveConfiguration/Segment:
    Shape = CIRCULAR
    SegmentReference = SEG_60
    SegmentSectorReference = SECTOR_SEG_60
    SegmentSectorDirection = Positive
    ElongationCompensation = UseAssemblySetting
    StopReaction = UseAssemblySetting
    SpeedFilter = UseAssemblySetting
8F1I01.BB4B.xxxx-1o : 8F1I01.BB4B.xxxx-1 v1.0.0.2  [PLK1 -> 8F1I01.AB2B.xxxx-1k.PLK2 [Cable Type=PowerlinkCable, Length=10, Version=1.0.0.3]; PLK2 -> 8F1I01.BB4B.xxxx-1t.PLK1 [Cable Type=PowerlinkCable, Length=10, Version=1.0.0.3]]
  EnableDNA = on
  DriveConfiguration:
    McTypeID = LLMConfig
  DriveConfiguration/Segment:
    Shape = CIRCULAR
    SegmentReference = SEG_40
    SegmentSectorReference = SECTOR_SEG_40
    SegmentSectorDirection = Positive
    ElongationCompensation = UseAssemblySetting
    StopReaction = UseAssemblySetting
    SpeedFilter = UseAssemblySetting
8F1I01.BB4B.xxxx-1p : 8F1I01.BB4B.xxxx-1 v1.0.0.2  [PLK1 -> 8F1I01.BB4B.xxxx-1q.PLK2 [Cable Type=PowerlinkCable, Length=10, Version=1.0.0.3]; PLK2 -> 8F1I01.BA2B.xxxx-1l.PLK1 [Cable Type=PowerlinkCable, Length=10, Version=1.0.0.3]]
  EnableDNA = on
  DriveConfiguration:
    McTypeID = LLMConfig
  DriveConfiguration/Segment:
    Shape = CIRCULAR
    SegmentReference = SEG_48
    SegmentSectorReference = SECTOR_SEG_48
    SegmentSectorDirection = Positive
    ElongationCompensation = UseAssemblySetting
    StopReaction = UseAssemblySetting
    SpeedFilter = UseAssemblySetting
8F1I01.BB4B.xxxx-1q : 8F1I01.BB4B.xxxx-1 v1.0.0.2  [PLK1 -> 8F1I01.BB4B.xxxx-1r.PLK2 [Cable Type=PowerlinkCable, Length=10, Version=1.0.0.3]; PLK2 -> 8F1I01.BB4B.xxxx-1p.PLK1 [Cable Type=PowerlinkCable, Length=10, Version=1.0.0.3]]
  EnableDNA = on
  DriveConfiguration:
    McTypeID = LLMConfig
  DriveConfiguration/Segment:
    Shape = CIRCULAR
    SegmentReference = SEG_47
    SegmentSectorReference = SECTOR_SEG_47
    SegmentSectorDirection = Positive
    ElongationCompensation = UseAssemblySetting
    StopReaction = UseAssemblySetting
    SpeedFilter = UseAssemblySetting
8F1I01.BB4B.xxxx-1r : 8F1I01.BB4B.xxxx-1 v1.0.0.2  [PLK1 -> 8F1I01.AB2B.xxxx-1l.PLK2 [Cable Type=PowerlinkCable, Length=10, Version=1.0.0.3]; PLK2 -> 8F1I01.BB4B.xxxx-1q.PLK1 [Cable Type=PowerlinkCable, Length=10, Version=1.0.0.3]]
  EnableDNA = on
  DriveConfiguration:
    McTypeID = LLMConfig
  DriveConfiguration/Segment:
    Shape = CIRCULAR
    SegmentReference = SEG_46
    SegmentSectorReference = SECTOR_SEG_46
    SegmentSectorDirection = Positive
    ElongationCompensation = UseAssemblySetting
    StopReaction = UseAssemblySetting
    SpeedFilter = UseAssemblySetting
8F1I01.BB4B.xxxx-1s : 8F1I01.BB4B.xxxx-1 v1.0.0.2  [PLK1 -> 8F1I01.BB4B.xxxx-1t.PLK2 [Cable Type=PowerlinkCable, Length=10, Version=1.0.0.3]; PLK2 -> 8F1I01.BA2B.xxxx-1k.PLK1 [Cable Type=PowerlinkCable, Length=10, Version=1.0.0.3]]
  EnableDNA = on
  DriveConfiguration:
    McTypeID = LLMConfig
  DriveConfiguration/Segment:
    Shape = CIRCULAR
    SegmentReference = SEG_42
    SegmentSectorReference = SECTOR_SEG_42
    SegmentSectorDirection = Positive
    ElongationCompensation = UseAssemblySetting
    StopReaction = UseAssemblySetting
    SpeedFilter = UseAssemblySetting
8F1I01.BB4B.xxxx-1t : 8F1I01.BB4B.xxxx-1 v1.0.0.2  [PLK1 -> 8F1I01.BB4B.xxxx-1o.PLK2 [Cable Type=PowerlinkCable, Length=10, Version=1.0.0.3]; PLK2 -> 8F1I01.BB4B.xxxx-1s.PLK1 [Cable Type=PowerlinkCable, Length=10, Version=1.0.0.3]]
  EnableDNA = on
  DriveConfiguration:
    McTypeID = LLMConfig
  DriveConfiguration/Segment:
    Shape = CIRCULAR
    SegmentReference = SEG_41
    SegmentSectorReference = SECTOR_SEG_41
    SegmentSectorDirection = Positive
    ElongationCompensation = UseAssemblySetting
    StopReaction = UseAssemblySetting
    SpeedFilter = UseAssemblySetting
8F1I01.BB4B.xxxx-1u : 8F1I01.BB4B.xxxx-1 v1.0.0.2  [PLK1 -> 8F1I01.BB4B.xxxx-1j.PLK2 [Cable Type=PowerlinkCable, Length=10, Version=1.0.0.3]; PLK2 -> 8F1I01.BA2B.xxxx-1f.PLK1 [Cable Type=PowerlinkCable, Length=10, Version=1.0.0.3]]
  EnableDNA = on
  DriveConfiguration:
    McTypeID = LLMConfig
  DriveConfiguration/Segment:
    Shape = CIRCULAR
    SegmentReference = SEG_53
    SegmentSectorReference = SECTOR_SEG_53
    SegmentSectorDirection = Positive
    ElongationCompensation = UseAssemblySetting
    StopReaction = UseAssemblySetting
    SpeedFilter = UseAssemblySetting
8F1I01.BB4B.xxxx-1v : 8F1I01.BB4B.xxxx-1 v1.0.0.2  [PLK1 -> 8F1I01.AB2B.xxxx-1m.PLK2 [Cable Type=PowerlinkCable, Length=10, Version=1.0.0.3]; PLK2 -> 8F1I01.BB4B.xxxx-1j.PLK1 [Cable Type=PowerlinkCable, Length=10, Version=1.0.0.3]]
  EnableDNA = on
  DriveConfiguration:
    McTypeID = LLMConfig
  DriveConfiguration/Segment:
    Shape = CIRCULAR
    SegmentReference = SEG_51
    SegmentSectorReference = SECTOR_SEG_51
    SegmentSectorDirection = Positive
    ElongationCompensation = UseAssemblySetting
    StopReaction = UseAssemblySetting
    SpeedFilter = UseAssemblySetting
8F1I01.BB4B.xxxx-1x : 8F1I01.BB4B.xxxx-1 v1.0.0.2  [PLK1 -> 8F1I01.AB2B.xxxx-1h.PLK2 [Cable Type=PowerlinkCable, Length=10, Version=1.0.0.3]; PLK2 -> 8F1I01.BA2B.xxxx-1h.PLK1 [Cable Type=PowerlinkCable, Length=10, Version=1.0.0.3]]
  EnableDNA = on
  DriveConfiguration:
    McTypeID = LLMConfig
  DriveConfiguration/Segment:
    Shape = CIRCULAR
    SegmentReference = SEG_66
    SegmentSectorReference = SECTOR_SEG_66
    SegmentSectorDirection = Positive
    ElongationCompensation = UseAssemblySetting
    StopReaction = UseAssemblySetting
    SpeedFilter = UseAssemblySetting
PC : PC_any v1.1.1.0 (OrderNumber=PC)
  ConfigurationID = Snapshot_Config1
  RemanentGlobalPvSize = 16000
  Cyclic1Duration = 10000
  Cyclic2Duration = 20000
  FileDevice1
  FileDeviceName1 = SvgData
  FileDevicePath1 = C:\projects\TrakSnapshot\Snapshot_V2\Logical
  FileDevice2
  FileDeviceName2 = SnapshotDevice
  FileDevicePath2 = C:\projects\TrakSnapshot\Snapshot_V2\Logical\Recipes
  ActivateOpcUa = 1
  OpcUaInformationModels_PV_Version = 1
```

### Config_1.assembly - PC/mappMotion/TrakOval/Config_1.assembly
```
Element gAssembly_1 (Type=assembly)
  Tracks:
    TrackSeparation = 0.030
    Track[1]:
      Segments:
        SegmentRef[1] = ::SEG_01
        SegmentRef[2] = ::SEG_02
        SegmentRef[3] = ::SEG_03
        SegmentRef[4] = ::SEG_04
        SegmentRef[5] = ::SEG_05
        SegmentRef[6] = ::SEG_06
        SegmentRef[7] = ::SEG_07
        SegmentRef[8] = ::SEG_08
        SegmentRef[9] = ::SEG_09
        SegmentRef[10] = ::SEG_10
        SegmentRef[11] = ::SEG_11
        SegmentRef[12] = ::SEG_12
        SegmentRef[13] = ::SEG_13
        SegmentRef[14] = ::SEG_14
        SegmentRef[15] = ::SEG_15
        SegmentRef[16] = ::SEG_16
        SegmentRef[17] = ::SEG_17
        SegmentRef[18] = ::SEG_18
        SegmentRef[19] = ::SEG_19
        SegmentRef[20] = ::SEG_20
      Position = Absolute
        SegmentRef = ::SEG_01
        SegmentCountDirection = RightToLeft
        Translation:
          X = 0.0
          Y = 0.0
          Z = 0.0
        Orientation:
          Angle1 = 0.0
          Angle2 = 0.0
          Angle3 = 180
    Track[2]:
      Segments:
        SegmentRef[1] = ::SEG_21
        SegmentRef[2] = ::SEG_22
        SegmentRef[3] = ::SEG_23
        SegmentRef[4] = ::SEG_24
        SegmentRef[5] = ::SEG_25
        SegmentRef[6] = ::SEG_26
        SegmentRef[7] = ::SEG_27
        SegmentRef[8] = ::SEG_28
        SegmentRef[9] = ::SEG_29
        SegmentRef[10] = ::SEG_30
        SegmentRef[11] = ::SEG_31
        SegmentRef[12] = ::SEG_32
        SegmentRef[13] = ::SEG_33
        SegmentRef[14] = ::SEG_34
        SegmentRef[15] = ::SEG_35
        SegmentRef[16] = ::SEG_36
        SegmentRef[17] = ::SEG_37
        SegmentRef[18] = ::SEG_38
      Position = RelativeToOne
        TrackSegmentPosition:
          SegmentRef = ::SEG_21
        Base:
          SegmentRef = ::SEG_11
          PositionRelativeTo = FromEnd
    Track[3]:
      Segments:
        SegmentRef[1] = ::SEG_39
        SegmentRef[2] = ::SEG_40
        SegmentRef[3] = ::SEG_41
        SegmentRef[4] = ::SEG_42
        SegmentRef[5] = ::SEG_43
        SegmentRef[6] = ::SEG_44
        SegmentRef[7] = ::SEG_45
        SegmentRef[8] = ::SEG_46
        SegmentRef[9] = ::SEG_47
        SegmentRef[10] = ::SEG_48
        SegmentRef[11] = ::SEG_49
      Position = RelativeToOne
        TrackSegmentPosition:
          SegmentRef = ::SEG_39
        Base:
          SegmentRef = ::SEG_25
          Position = 0.330
    Track[4]:
      Segments:
        SegmentRef[1] = ::SEG_50
        SegmentRef[2] = ::SEG_51
        SegmentRef[3] = ::SEG_52
        SegmentRef[4] = ::SEG_53
        SegmentRef[5] = ::SEG_54
      Position = RelativeToOne
        TrackSegmentPosition:
          SegmentRef = ::SEG_54
          PositionRelativeTo = FromEnd
        Base:
          SegmentRef = ::SEG_14
    Track[5]:
      Segments:
        SegmentRef[1] = ::SEG_55
        SegmentRef[2] = ::SEG_56
        SegmentRef[3] = ::SEG_57
        SegmentRef[4] = ::SEG_58
      Position = RelativeToOne
        TrackSegmentPosition:
          SegmentRef = ::SEG_55
          PositionRelativeTo = FromEnd
        Base:
          SegmentRef = ::SEG_50
    Track[6]:
      Segments:
        SegmentRef[1] = ::SEG_59
        SegmentRef[2] = ::SEG_60
        SegmentRef[3] = ::SEG_61
      Position = RelativeToOne
        TrackSegmentPosition:
          SegmentRef = ::SEG_59
        Base:
          SegmentRef = ::SEG_05
          PositionRelativeTo = FromEnd
    Track[7]:
      Segments:
        SegmentRef[1] = ::SEG_62
        SegmentRef[2] = ::SEG_63
        SegmentRef[3] = ::SEG_64
      Position = RelativeToOne
        TrackSegmentPosition:
          SegmentRef = ::SEG_62
        Base:
          SegmentRef = ::SEG_61
          PositionRelativeTo = FromEnd
    Track[8]:
      Segments:
        SegmentRef[1] = ::SEG_65
        SegmentRef[2] = ::SEG_66
        SegmentRef[3] = ::SEG_67
      Position = RelativeToOne
        TrackSegmentPosition:
          SegmentRef = ::SEG_65
        Base:
          SegmentRef = ::SEG_02
          PositionRelativeTo = FromEnd
    Track[9]:
      Segments:
        SegmentRef[1] = ::SEG_68
        SegmentRef[2] = ::SEG_69
        SegmentRef[3] = ::SEG_70
      Position = RelativeToOne
        TrackSegmentPosition:
          SegmentRef = ::SEG_68
        Base:
          SegmentRef = ::SEG_67
          PositionRelativeTo = FromEnd
  CommonSegmentSettings:
    SegmentSimulationOnPLC = Off
    ElongationCompensation = Inactive
    StopReaction = InductionHalt
    SpeedFilter = NotUsed
    ControllerParameters:
      DefaultParameter:
        Controller:
          Position:
            ProportionalGain = 200
          Speed:
            ProportionalGain = 80
            IntegrationTime = 0.0
          FeedForward:
            TotalMass = 1
            ForcePositive = 0.0
            ForceNegative = 0.0
            SpeedForceFactor = 0.0
            ForceLoad = 0.0
        MovementErrorLimits:
          PositionError = 0.001
          VelocityError = 0.05
      AdditionalParameterSets = NotUsed
    ScopeOfErrorReaction = Assembly
    ShuttleIdentificationTime = 0
  Shuttles:
    MaxShuttleCount = 100
    DistanceReserve:
      Collision = 0.001
      ErrorStop = 0.005
    ShuttleStereotypes:
      ShuttleStRef[1] = ShuttleStereotype_1
    MagnetPlateConfigurations:
      ShuttleType[1] = 8F1SA.100.xxxxxx-x
    CollisionAvoidance:
      Strategy = Constant
      MaximumModelDimensions:
        Length:
          ExtentToFront = 0.025
          ExtentToBack = 0.025
        Width:
          Width = 0.025
  AssemblyFeatures:
    AssemblyFeatureRef[1] = AssemblyFeature_1
  Visualization:
    MonitoringPv = gShuttleMon
    ProcessingTaskClass = 2
```

### Config_2.shuttlestereotype - PC/mappMotion/TrakOval/Config_2.shuttlestereotype
```
Element ShuttleStereotype_1 (Type=shuttlestereotype)
  MeasurementUnit = 5067858
  MeasurementResolution = 0.00001
  MovementLimits = Internal
    VelocityIsReadOnly = 0
    Velocity:
      Velocity = 4
    AccelerationIsReadOnly = 0
    Acceleration:
      Acceleration = 40
    DecelerationIsReadOnly = 0
    Deceleration:
      Deceleration = 40
    UpdateMode = Immediately
  JerkFilter = NotUsed
  UserData:
    Size = 20
```

### Config_3.sector - PC/mappMotion/TrakOval/Config_3.sector
```
Element Spawn_Sector (Type=sector)
  Type = Composed
    StartSegment:
      SegmentRef = ::SEG_01
    IntermediateSegments:
      SegmentRef[1] = ::SEG_02
      SegmentRef[2] = ::SEG_03
      SegmentRef[3] = ::SEG_04
      SegmentRef[4] = ::SEG_05
      SegmentRef[5] = ::SEG_06
      SegmentRef[6] = ::SEG_07
      SegmentRef[7] = ::SEG_08
      SegmentRef[8] = ::SEG_09
      SegmentRef[9] = ::SEG_10
      SegmentRef[10] = ::SEG_11
      SegmentRef[11] = ::SEG_12
      SegmentRef[12] = ::SEG_13
      SegmentRef[13] = ::SEG_14
      SegmentRef[14] = ::SEG_15
      SegmentRef[15] = ::SEG_16
      SegmentRef[16] = ::SEG_17
      SegmentRef[17] = ::SEG_18
      SegmentRef[18] = ::SEG_19
    EndSegment:
      SegmentRef = ::SEG_20
      PositionRelativeTo = FromEnd
Element Load_Unload_Sector (Type=sector)
  Type = Composed
    StartSegment:
      SegmentRef = ::SEG_44
    EndSegment:
      SegmentRef = ::SEG_44
      Position = 0.330
Element Process_1_Sector (Type=sector)
  Type = Composed
    StartSegment:
      SegmentRef = ::SEG_18
    EndSegment:
      SegmentRef = ::SEG_18
      Position = 0.120
Element Process_2_Sector (Type=sector)
  Type = Composed
    StartSegment:
      SegmentRef = ::SEG_30
      PositionRelativeTo = FromEnd
    EndSegment:
      SegmentRef = ::SEG_30
      Position = 0.330
      PositionRelativeTo = FromEnd
Element Process_3_Sector (Type=sector)
  Type = Composed
    StartSegment:
      SegmentRef = ::SEG_56
    EndSegment:
      SegmentRef = ::SEG_56
      Position = 0.225
Element Reject_LeftUp (Type=sector)
  Type = Composed
    StartSegment:
      SegmentRef = ::SEG_70
      PositionRelativeTo = FromEnd
    IntermediateSegments:
      SegmentRef[1] = ::SEG_69
    EndSegment:
      SegmentRef = ::SEG_68
      Position = 0
Element Reject_RightUp (Type=sector)
  Type = Composed
    StartSegment:
      SegmentRef = ::SEG_67
    EndSegment:
      SegmentRef = ::SEG_67
      Position = 0
      PositionRelativeTo = FromEnd
Element Reject_RightDown (Type=sector)
  Type = Composed
    StartSegment:
      SegmentRef = ::SEG_67
      PositionRelativeTo = FromEnd
    IntermediateSegments:
      SegmentRef[1] = ::SEG_66
    EndSegment:
      SegmentRef = ::SEG_65
      Position = 0
Element Flipper_LeftUp (Type=sector)
  Type = Composed
    StartSegment:
      SegmentRef = ::SEG_64
      PositionRelativeTo = FromEnd
    IntermediateSegments:
      SegmentRef[1] = ::SEG_63
    EndSegment:
      SegmentRef = ::SEG_62
      Position = 0
Element Flipper_RightUp (Type=sector)
  Type = Composed
    StartSegment:
      SegmentRef = ::SEG_61
    EndSegment:
      SegmentRef = ::SEG_61
      Position = 0
      PositionRelativeTo = FromEnd
Element Flipper_RightDown (Type=sector)
  Type = Composed
    StartSegment:
      SegmentRef = ::SEG_61
      PositionRelativeTo = FromEnd
    IntermediateSegments:
      SegmentRef[1] = ::SEG_60
    EndSegment:
      SegmentRef = ::SEG_59
      Position = 0
```

### Config_4.assemblyfeature - PC/mappMotion/TrakOval/Config_4.assemblyfeature
```
Element AssemblyFeature_1 (Type=assemblyfeature)
  Type = InitShuttleSim
    InitShuttleSim[1]:
      SectorRef = Spawn_Sector
      Orientation = Positive
      ShuttleDefinition = ShuttleSetDefinition
        StartPosition = 0.0
        NumberOfShuttles = 50
        DistnaceBetweenShuttles = 0.05
```

### Config_5.processpointlist - PC/mappMotion/TrakOval/Config_5.processpointlist
```
Element PP_List (Type=processpointlist)
  ProcessPoint[0]:
    Name = PP_Load_Unload
    SectorRef = Load_Unload_Sector
    TriggerEventBufferSize = 10
    BarrierFunctionality = Off
  ProcessPoint[1]:
    Name = PP_Process_1
    SectorRef = Process_1_Sector
    TriggerEventBufferSize = 10
    BarrierFunctionality = Off
  ProcessPoint[2]:
    Name = PP_Process_2
    SectorRef = Process_2_Sector
    TriggerEventBufferSize = 10
    BarrierFunctionality = Off
  ProcessPoint[3]:
    Name = PP_Process_3
    SectorRef = Process_3_Sector
    TriggerEventBufferSize = 10
    BarrierFunctionality = Off
  ProcessPoint[4]:
    Name = PP_Reject
    SectorRef = Reject_LeftUp
    Position = 0.915
    TriggerEventBufferSize = 10
    BarrierFunctionality = Off
  ProcessPoint[5]:
    Name = PP_Flipper
    SectorRef = Flipper_LeftUp
    Position = 0.915
    TriggerEventBufferSize = 10
    BarrierFunctionality = Off
  ProcessPoint[6]:
    Name = PP_RejectEntrance
    SectorRef = Reject_LeftUp
    Position = 0.57
    TriggerEventBufferSize = 10
    BarrierFunctionality = On
  ProcessPoint[7]:
    Name = PP_RejectExit
    SectorRef = Reject_RightDown
    Position = 0.57
    TriggerEventBufferSize = 10
    BarrierFunctionality = Off
  ProcessPoint[8]:
    Name = PP_FlipperEntrance
    SectorRef = Flipper_LeftUp
    Position = 0.57
    TriggerEventBufferSize = 10
    BarrierFunctionality = On
  ProcessPoint[9]:
    Name = PP_FlipperExit
    SectorRef = Flipper_RightDown
    Position = 0.57
    TriggerEventBufferSize = 10
    BarrierFunctionality = Off
```

## Logical view

Binary libraries used (declarations not repeated): operator, runtime, astime, AsIecCon, McBase, McAxis, McAcpTrak, MpAxis, MpBase, McAcpAx, AsBrStr, standard, MpRecipe, sys_lib, AsBrMath

### Global.var - Global variables
```iecst
VAR
	gShuttleMon : McAcpTrakAssemblyMonData;
END_VAR
VAR RETAIN
	gDEV_SnapshotStructure : TrakSnap_type;
END_VAR
VAR
	gPowerOn : BOOL;
	gTrakRunning : BOOL;
END_VAR
```

### Package Logical/Libraries - Global libraries

### Library Logical/Libraries/TrakSnap (IEC)

#### Types.typ - Exported data types
```iecst
(*User Structure for Snapshot*)

TYPE
	TrakSnap_type : 	STRUCT
		UserData : ARRAY[0..TRAKSNAP_NUM_SHUTTLES]OF UserDataTyp; (*User data for the shuttles*)
		SegmentInfo : ARRAY[0..TRAKSNAP_NUM_SHUTTLES]OF SegmentInfo_type; (*Position and orientation output from the ShReadSecPos FUB*)
		ShuttleInfo : ARRAY[0..TRAKSNAP_NUM_SHUTTLES]OF ShuttleInfo_type; (*Abbreviated output of the ShReadInfo FUB*)
	END_STRUCT;
END_TYPE

(**)
(*Shuttle User Data*)

TYPE
	UserDataTyp : 	STRUCT  (*User data structure*)
		Color : UserColorEnum; (*Shuttle colour*)
		ShuttleID : UINT; (*Shuttle ID*)
		StationNum : USINT; (*Station number *)
		ShuttleSerialNum : ARRAY[0..11]OF USINT; (*Shuttle serial number*)
	END_STRUCT;
	UserColorEnum :
		( (*Shuttle colours*)
		GRAY := 0,
		BLUE := 1,
		RED := 2,
		GREEN := 3,
		YELLOW := 4,
		ORANGE := 5
		);
END_TYPE

(**)
(*An abbreviated segment info structure*)

TYPE
	SegmentInfo_type : 	STRUCT
		CurrentPosition : ARRAY[0..3]OF LREAL;
		CurrentSegment : ARRAY[0..3]OF STRING[32];
	END_STRUCT;
END_TYPE

(**)
(*An abbreviated shuttle info structure*)

TYPE
	ShuttleInfo_type : 	STRUCT
		CurrentPosition : LREAL;
		CurrentSector : STRING[32];
		CurrentVelocity : REAL;
		TargetPosition : LREAL;
		TargetSector : STRING[32];
		VelocityAtDestination : REAL;
	END_STRUCT;
END_TYPE

(**)
(*Internal Structure for SnapshotTaker FUB*)

TYPE
	TrakSnapCapInternal_type : 	STRUCT
		State : TrakSnapCapState_enum;
		FB : TrakSnapCapInternalFB_type;
		Shuttles : ARRAY[0..TRAKSNAP_NUM_SHUTTLES]OF McAxisType;
		Index : UINT;
		CountRemaining : UINT;
		CurrentDateTime : DATE_AND_TIME;
		CurrentDateTime_Str : STRING[100];
	END_STRUCT;
	TrakSnapCapState_enum :
		(
		SNAPCAP_IDLE,
		SNAPCAP_GET_SHUTTLES,
		SNAPCAP_CHECK_REMAINING_COUNT,
		SNAPCAP_READY,
		SNAPCAP_CAPTURE,
		SNAPCAP_SAVE,
		SNAPCAP_DONE,
		SNAPCAP_RESET,
		SNAPCAP_ERROR
		);
	TrakSnapCapInternalFB_type : 	STRUCT
		AsmGetShuttle : MC_BR_AsmGetShuttle_AcpTrak;
		ShCopyUserData : ARRAY[0..TRAKSNAP_NUM_SHUTTLES]OF MC_BR_ShCopyUserData_AcpTrak;
		ShReadSegmentInfo : ARRAY[0..TRAKSNAP_NUM_SHUTTLES]OF MC_BR_ShReadSegmentInfo_AcpTrak;
		ShReadInfo : ARRAY[0..TRAKSNAP_NUM_SHUTTLES]OF MC_BR_ShReadInfo_AcpTrak;
		RecipeXML : MpRecipeXml;
		RecipeRegPar : MpRecipeRegPar;
		GetTime : DTGetTime;
		DTRecipeConverter : EpochConverter;
	END_STRUCT;
END_TYPE

(**)
(*Internal Structure for SnapshotSpawner FUB*)

TYPE
	TrakSnapSpawnInternal_type : 	STRUCT
		State : TrakSnapSpawnState_enum;
		FB : TrakSnapSpawnInternalFB_type;
		Shuttles : ARRAY[0..TRAKSNAP_NUM_SHUTTLES]OF McAxisType;
		Index : UINT;
		SegmentSector : SegmentSector_type;
		SectorReference : UDINT;
		SectorReferenceSize : UDINT;
		PV_XGETADR_ERROR_ID : UINT;
	END_STRUCT;
	TrakSnapSpawnState_enum :
		(
		SNAPSPAWN_IDLE,
		SNAPSPAWN_READY,
		SNAPSPAWN_LOAD_RECIPE,
		SNAPSPAWN_PICK_SEGSEC,
		SNAPSPAWN_SPAWN_SHUTTLE,
		SNAPSPAWN_SET_USERDATA,
		SNAPSPAWN_DONE,
		SNAPSPAWN_RESET,
		SNAPSPAWN_ERROR
		);
	TrakSnapSpawnInternalFB_type : 	STRUCT
		SecAddShuttle : MC_BR_SecAddShuttle_AcpTrak;
		ShCopyUserData : MC_BR_ShCopyUserData_AcpTrak;
		RecipeXML : MpRecipeXml;
		RecipeRegPar : MpRecipeRegPar;
	END_STRUCT;
	SegmentSector_type : 	STRUCT
		Prefix : STRING[8] := 'SECTOR_';
		Name : STRING[32];
		Index : USINT;
		BestOption : USINT;
		Valid : ARRAY[0..3]OF BOOL;
		Position : ARRAY[0..3]OF LREAL;
	END_STRUCT;
END_TYPE
```

#### Constants.var - Exported constants
```iecst
(*TRAK SNAP*)
VAR CONSTANT
	TRAKSNAP_NUM_SHUTTLES : UINT := 50;
END_VAR
(**)
(*SNAP CAP*)
(*Error Numbers*)
VAR CONSTANT
	CAP_RECIPE_INIT_FAILED : DINT := -60000; (*Error when enabling the recipe FUBs*)
	CAP_GET_SHUTTLES_FAILED : DINT := -60001; (*Error with the AsmGetShuttle FUB*)
	CAP_TOO_MANY_SHUTTLES : DINT := -60002; (*TotalCount > TRAKSNAP_NUM_SHUTTLES. Config is higher than library constant*)
	CAP_READ_SEGMENT_INFO_FAILED : DINT := -61000; (*Error with ShReadSectorPos FUB. The index of the shuttle will be added to -61000 for better troubleshooting.*)
	CAP_READ_SHUTTLE_INFO_FAILED : DINT := -62000; (*Error with ShReadInfo FUB. The index of the shuttle will be added to -62000 for better troubleshooting.*)
	CAP_GET_USERDATA_FAILED : DINT := -63000; (*Error with ShCopyUserData FUB. The index of the shuttle will be added to -63000 for better troubleshooting.*)
	CAP_SAVE_RECIPE_FAILED : DINT := -60003; (*Error on the recipe FUBs when saving the recipe*)
END_VAR
(**)
(*SNAP SPAWN*)
(*Error Numbers*)
VAR CONSTANT
	SPAWN_RECIPE_INIT_FAILED : DINT := -60004; (*Error when enabling the recipe FUBs*)
	SPAWN_SNAPSHOT_TO_LOAD_EMPTY : DINT := -60005; (*The parameter "SnapshotToLoad" is empty*)
	SPAWN_LOAD_RECIPE_FAILED : DINT := -60006; (*Error on the recipe FUBs when loading the recipe*)
	SPAWN_NO_POS_FOR_SHUTTLE_SPAWN : DINT := -64000; (*ShReadInfo and ShReadSegmentInfo both lacked references. The index of the shuttle will be added to -64000 for better troubleshooting.*)
	SPAWN_ADD_SHUTTLE_FAILED : DINT := -65000; (*Error with SecAddShuttle FUB. The index of the shuttle will be added to -64000 for better troubleshooting.*)
	SPAWN_SET_USERDATA_FAILED : DINT := -66000; (*Error with ShCopyUserData FUB. The index of the shuttle will be added to -65000 for better troubleshooting.*)
END_VAR
(**)
(*EPOCH CONVERTER*)
VAR CONSTANT
	EPOCH_OFFSET : DINT := 0; (*Past Values: 24513, -48657, -24144*)
END_VAR
```

#### TrakSnap.fun - Exported functions and function blocks
```iecst
FUNCTION_BLOCK TrakSnapCap (*Function block that captures all spawned shuttles and their data*)
	VAR_INPUT
		Enable : BOOL;
		Capture : BOOL;
		Assembly : REFERENCE TO McAssemblyType; (*Assembly to capture startup data*)
		TrakSnapStructure : REFERENCE TO TrakSnap_type;
		TrakSnapStructureName : {REDUND_UNREPLICABLE} STRING[100];
		RecipeLink : REFERENCE TO MpComIdentType;
	END_VAR
	VAR_OUTPUT
		Active : BOOL;
		Ready : BOOL;
		Busy : BOOL;
		Done : BOOL;
		NumShuttlesFound : UINT;
		Error : BOOL; (*Error present on diagnostic function*)
		ErrorID : DINT; (*Error ID of current error*)
	END_VAR
	VAR
		Internal : TrakSnapCapInternal_type; (*Internal datatype*)
	END_VAR
END_FUNCTION_BLOCK

FUNCTION_BLOCK TrakSnapSpawn (*Function block that spawns all shuttles and their data from a saved snapshot*)
	VAR_INPUT
		Enable : BOOL;
		Spawn : BOOL;
		TrakSnapStructure : REFERENCE TO TrakSnap_type;
		TrakSnapStructureName : {REDUND_UNREPLICABLE} STRING[100];
		RecipeLink : REFERENCE TO MpComIdentType;
		SnapshotToLoad : STRING[100];
		NumShuttles : UINT;
	END_VAR
	VAR_OUTPUT
		Active : BOOL;
		Ready : BOOL;
		Done : BOOL;
		Busy : BOOL;
		Error : BOOL; (*Error present on diagnostic function*)
		ErrorID : DINT; (*Error ID of current error*)
	END_VAR
	VAR
		Internal : TrakSnapSpawnInternal_type; (*Internal datatype*)
	END_VAR
END_FUNCTION_BLOCK

FUNCTION_BLOCK EpochConverter (*Converts epoch time to STR of format similar to DT but without the ":" character.*)
	VAR_INPUT
		Input : {REDUND_UNREPLICABLE} UDINT;
		Offset : {REDUND_UNREPLICABLE} DINT;
		Execute : BOOL;
	END_VAR
	VAR_OUTPUT
		DTString_For_Recipe : STRING[100];
	END_VAR
	VAR
		InternalState : USINT;
		Year : {REDUND_UNREPLICABLE} UDINT;
		Year_Str : {REDUND_UNREPLICABLE} STRING[5];
		Month : {REDUND_UNREPLICABLE} UDINT;
		Month_Str : {REDUND_UNREPLICABLE} STRING[5];
		Day : {REDUND_UNREPLICABLE} UDINT;
		Day_Str : {REDUND_UNREPLICABLE} STRING[5];
		Hour : {REDUND_UNREPLICABLE} UDINT;
		Hour_Str : {REDUND_UNREPLICABLE} STRING[5];
		Minute : {REDUND_UNREPLICABLE} UDINT;
		Minute_Str : {REDUND_UNREPLICABLE} STRING[5];
		Second : {REDUND_UNREPLICABLE} UDINT;
		Second_Str : {REDUND_UNREPLICABLE} STRING[5];
		Remainder : {REDUND_UNREPLICABLE} UDINT;
		DateWord : {REDUND_UNREPLICABLE} STRING[5] := 'date';
		TimeWord : {REDUND_UNREPLICABLE} STRING[5] := 'time';
		SpaceCharacter : {REDUND_UNREPLICABLE} STRING[2] := ' ';
		UnderscoreCharacter : {REDUND_UNREPLICABLE} STRING[2] := '_';
	END_VAR
END_FUNCTION_BLOCK
```

#### TrakSnapCap.st - StarSync Implementation
```iecst
(*********************************************************************************
 * Copyright: B&R Industrial Automation GmbH
 * Author:    nealj
 * Created:   October 18, 2021/11:10 AM
 * The SnapshotTaker FUB will gather the list of shuttles and monitor their
 * postions when enabled. When execute is TRUE, the FUB will gather the user data
 * and shuttle info of each shuttle.
 *
 * NOTE: The FUB works on the assumption that a global trak sector has been
 * created. This is a sector that encompasses the entire assembly in one
 * continuous path. Overlap is allowed.
 *********************************************************************************)

FUNCTION_BLOCK TrakSnapCap

	Internal.FB.GetTime.enable          := Enable;
	Internal.CurrentDateTime            := Internal.FB.GetTime.DT1;
	Internal.FB.DTRecipeConverter.Input := DT_TO_UDINT(Internal.CurrentDateTime);
	IF (Enable AND NOT Internal.FB.DTRecipeConverter.Execute) THEN
		Internal.FB.DTRecipeConverter.Execute := TRUE;
	END_IF
	Internal.CurrentDateTime_Str        := Internal.FB.DTRecipeConverter.DTString_For_Recipe;

	Internal.FB.RecipeXML.Enable     := Enable;
	Internal.FB.RecipeXML.MpLink     := ADR(RecipeLink);
	Internal.FB.RecipeXML.DeviceName := ADR('SnapshotDevice');
	Internal.FB.RecipeXML.FileName   := ADR(Internal.CurrentDateTime_Str);

	Internal.FB.RecipeRegPar.Enable := Internal.FB.RecipeXML.Active;
	Internal.FB.RecipeRegPar.MpLink := ADR(RecipeLink);
	Internal.FB.RecipeRegPar.PVName := ADR(TrakSnapStructureName);

	CASE Internal.State OF
		//************************************************************************************************************
		SNAPCAP_IDLE:
			IF (Internal.FB.RecipeXML.Error OR Internal.FB.RecipeRegPar.Error) THEN
				//RECIPE INIT FAILED
				Error          := TRUE;
				ErrorID        := CAP_RECIPE_INIT_FAILED;
				Internal.State := SNAPCAP_ERROR;
			ELSIF (Enable AND Internal.FB.RecipeXML.Active AND Internal.FB.RecipeRegPar.Active) THEN
				//Set the active flag, clear the user structure and shuttle list, and start the AsmGetShuttle FUB
				Active                             := TRUE;
				brsmemset(ADR(TrakSnapStructure),0,SIZEOF(TrakSnapStructure));
				brsmemset(ADR(Internal.Shuttles),0,SIZEOF(Internal.Shuttles));
				Internal.FB.AsmGetShuttle.Assembly := ADR(Assembly);
				Internal.FB.AsmGetShuttle.Enable   := TRUE;
				Internal.Index                     := 0;
				Internal.State                     := SNAPCAP_GET_SHUTTLES;
			END_IF

		//************************************************************************************************************
		SNAPCAP_GET_SHUTTLES:
			IF NOT Enable THEN
				Internal.State := SNAPCAP_RESET;
			ELSIF Internal.FB.AsmGetShuttle.Error THEN
				//GET SHUTTLES FAILED
				Error          := TRUE;
				ErrorID        := CAP_GET_SHUTTLES_FAILED;
				Internal.State := SNAPCAP_ERROR;
			ELSIF (Internal.FB.AsmGetShuttle.Valid AND (Internal.Shuttles[Internal.Index].controlif = 0)) THEN
				IF (Internal.FB.AsmGetShuttle.TotalCount > TRAKSNAP_NUM_SHUTTLES) THEN
					//TOO MANY SHUTTLES
					Error          := TRUE;
					ErrorID        := CAP_TOO_MANY_SHUTTLES;
					Internal.State := SNAPCAP_ERROR;
				ELSE
					//Update the list of shuttles
					Internal.FB.AsmGetShuttle.Next    := FALSE;
					Internal.Shuttles[Internal.Index] := Internal.FB.AsmGetShuttle.Axis;
					Internal.Index                    := Internal.Index + 1;
					Internal.State                    := SNAPCAP_CHECK_REMAINING_COUNT;
				END_IF
			END_IF

		//************************************************************************************************************
		SNAPCAP_CHECK_REMAINING_COUNT:
			IF NOT Enable THEN
				Internal.State := SNAPCAP_RESET;
			ELSIF Internal.FB.AsmGetShuttle.RemainingCount > 0 THEN
				Internal.FB.AsmGetShuttle.Next := TRUE;
				Internal.State                 := SNAPCAP_GET_SHUTTLES;
			ELSE
				//Update the count, and configure the ShReadSegmentInfo & ShReadInfo FUBs
				NumShuttlesFound := Internal.FB.AsmGetShuttle.TotalCount;
				FOR Internal.Index:=0 TO (NumShuttlesFound-1) DO
					Internal.FB.ShReadSegmentInfo[Internal.Index].Axis   := ADR(Internal.Shuttles[Internal.Index]);
					Internal.FB.ShReadSegmentInfo[Internal.Index].Enable := TRUE;
					Internal.FB.ShReadInfo[Internal.Index].Axis          := ADR(Internal.Shuttles[Internal.Index]);
					Internal.FB.ShReadInfo[Internal.Index].Enable        := TRUE;
				END_FOR
				Ready          := TRUE;
				Internal.State := SNAPCAP_READY;
			END_IF

		//************************************************************************************************************
		SNAPCAP_READY:
			//ADD CONDITION TO DISABLE WHEN ENABLE IS RESET
			IF NOT Enable THEN
				Internal.State := SNAPCAP_RESET;
			ELSIF Internal.FB.AsmGetShuttle.TotalCount <> NumShuttlesFound THEN
				//If the shuttle count of the AsmGetShuttle FUB changes, clear the user structure and shuttle list and update the shuttle list
				FOR Internal.Index:=0 TO (TRAKSNAP_NUM_SHUTTLES) DO
					Internal.FB.ShReadSegmentInfo[Internal.Index].Enable := FALSE;
					Internal.FB.ShReadInfo[Internal.Index].Enable        := FALSE;
				END_FOR
				brsmemset(ADR(TrakSnapStructure),0,SIZEOF(TrakSnapStructure));
				brsmemset(ADR(Internal.Shuttles),0,SIZEOF(Internal.Shuttles)); //Is this the proper way to clear the array? -JRN 10/18/21
				Internal.Index                     := 0;
				Internal.State                     := SNAPCAP_GET_SHUTTLES;
			ELSIF Capture THEN
				//When the capture command is set, leave the state to capture the data and info
				Ready                                  := FALSE;
				Busy                                   := TRUE;
				Internal.Index                         := 0;
				FOR Internal.Index:=0 TO (NumShuttlesFound-1) DO
					Internal.FB.ShCopyUserData[Internal.Index].Axis        := ADR(Internal.Shuttles[Internal.Index]);
					Internal.FB.ShCopyUserData[Internal.Index].DataAddress := ADR(TrakSnapStructure.UserData[Internal.Index]);
					Internal.FB.ShCopyUserData[Internal.Index].DataSize    := SIZEOF(TrakSnapStructure.UserData[Internal.Index]);
					Internal.FB.ShCopyUserData[Internal.Index].Execute     := TRUE;
				END_FOR
				Internal.State                         := SNAPCAP_CAPTURE;
			ELSE
				//Check the ShReadSegmentInfo and ShReadInfo FUBs for errors
				FOR Internal.Index:=0 TO (NumShuttlesFound-1) DO
					IF Internal.FB.ShReadSegmentInfo[Internal.Index].Error THEN
						//READ GLOBAL POS FAILED
						Error          := TRUE;
						ErrorID        := CAP_READ_SEGMENT_INFO_FAILED + Internal.Index;
						Internal.State := SNAPCAP_ERROR;
					ELSIF Internal.FB.ShReadInfo[Internal.Index].Error THEN
						//READ SHUTTLE INFO FAILED
						Error          := TRUE;
						ErrorID        := CAP_READ_SHUTTLE_INFO_FAILED + Internal.Index;
						Internal.State := SNAPCAP_ERROR;
					END_IF
				END_FOR
			END_IF

			//************************************************************************************************************
		SNAPCAP_CAPTURE:
			FOR Internal.Index:=0 TO (NumShuttlesFound-1) DO
				IF Internal.FB.ShCopyUserData[Internal.Index].Error THEN
					//GET USERDATA FAILED
					Error          := TRUE;
					ErrorID        := CAP_GET_USERDATA_FAILED + Internal.Index;
					Internal.State := SNAPCAP_ERROR;
				ELSIF Internal.FB.ShCopyUserData[Internal.Index].Done THEN
					Internal.FB.ShCopyUserData[Internal.Index].Execute                  := FALSE;
					//Read in segment information. A shuttle can be on up to 4 segments at once, so all possibilities are gathered
					TrakSnapStructure.SegmentInfo[Internal.Index].CurrentPosition[0]    := Internal.FB.ShReadSegmentInfo[Internal.Index].SegmentInfo.SegmentCurrentValues[0].Position;
					TrakSnapStructure.SegmentInfo[Internal.Index].CurrentSegment[0]     := Internal.FB.ShReadSegmentInfo[Internal.Index].SegmentInfo.SegmentCurrentValues[0].SegmentName;
					TrakSnapStructure.SegmentInfo[Internal.Index].CurrentPosition[1]    := Internal.FB.ShReadSegmentInfo[Internal.Index].SegmentInfo.SegmentCurrentValues[1].Position;
					TrakSnapStructure.SegmentInfo[Internal.Index].CurrentSegment[1]     := Internal.FB.ShReadSegmentInfo[Internal.Index].SegmentInfo.SegmentCurrentValues[1].SegmentName;
					TrakSnapStructure.SegmentInfo[Internal.Index].CurrentPosition[2]    := Internal.FB.ShReadSegmentInfo[Internal.Index].SegmentInfo.SegmentCurrentValues[2].Position;
					TrakSnapStructure.SegmentInfo[Internal.Index].CurrentSegment[2]     := Internal.FB.ShReadSegmentInfo[Internal.Index].SegmentInfo.SegmentCurrentValues[2].SegmentName;
					TrakSnapStructure.SegmentInfo[Internal.Index].CurrentPosition[3]    := Internal.FB.ShReadSegmentInfo[Internal.Index].SegmentInfo.SegmentCurrentValues[3].Position;
					TrakSnapStructure.SegmentInfo[Internal.Index].CurrentSegment[3]     := Internal.FB.ShReadSegmentInfo[Internal.Index].SegmentInfo.SegmentCurrentValues[3].SegmentName;
					//Read in shuttle information
					TrakSnapStructure.ShuttleInfo[Internal.Index].CurrentPosition       := Internal.FB.ShReadInfo[Internal.Index].ShuttleInfo.CurrentValues.ActualModuloPosition;
					TrakSnapStructure.ShuttleInfo[Internal.Index].CurrentSector         := Internal.FB.ShReadInfo[Internal.Index].ShuttleInfo.CurrentValues.SectorName;
					TrakSnapStructure.ShuttleInfo[Internal.Index].CurrentVelocity       := Internal.FB.ShReadInfo[Internal.Index].ShuttleInfo.CurrentValues.Velocity;
					TrakSnapStructure.ShuttleInfo[Internal.Index].TargetPosition        := Internal.FB.ShReadInfo[Internal.Index].ShuttleInfo.RouteDestinationInfo.Position;
					TrakSnapStructure.ShuttleInfo[Internal.Index].TargetSector          := Internal.FB.ShReadInfo[Internal.Index].ShuttleInfo.RouteDestinationInfo.SectorName;
					TrakSnapStructure.ShuttleInfo[Internal.Index].VelocityAtDestination := Internal.FB.ShReadInfo[Internal.Index].ShuttleInfo.RouteDestinationInfo.VelocityAtDestination;
				END_IF
			END_FOR
			IF NOT Enable THEN
				Internal.State := SNAPCAP_RESET;
			ELSIF NOT Error THEN
				Internal.FB.RecipeXML.Save := TRUE;
				Internal.State             := SNAPCAP_DONE;
			END_IF

			//************************************************************************************************************
		SNAPCAP_DONE:
			IF (Internal.FB.RecipeXML.Error OR Internal.FB.RecipeRegPar.Error) THEN
				//SAVE RECIPE FAILED
				Error          := TRUE;
				ErrorID        := CAP_SAVE_RECIPE_FAILED;
				Internal.State := SNAPCAP_ERROR;
			ELSIF (Internal.FB.RecipeXML.CommandDone AND NOT Done) THEN
				Busy := FALSE;
				Done := TRUE;
			ELSIF NOT Capture THEN
				Done           := FALSE;
				Ready          := TRUE;
				Internal.State := SNAPCAP_READY;
			ELSIF NOT Enable THEN
				Internal.State := SNAPCAP_RESET;
			END_IF

		//************************************************************************************************************
		SNAPCAP_RESET:
			Active  := FALSE;
			Ready   := FALSE;
			Capture := FALSE;
			Busy    := FALSE;
			Done    := FALSE;
			Active  := FALSE;
			Error   := FALSE;
			ErrorID := 0;

            Internal.FB.AsmGetShuttle.Enable                     := FALSE;
			FOR Internal.Index:=0 TO TRAKSNAP_NUM_SHUTTLES DO
			Internal.FB.ShReadSegmentInfo[Internal.Index].Enable := FALSE;
			Internal.FB.ShCopyUserData[Internal.Index].Execute   := FALSE;
			Internal.FB.ShReadInfo[Internal.Index].Enable        := FALSE;
			END_FOR

			Internal.Index := 0;
			Internal.State := SNAPCAP_IDLE;

		//************************************************************************************************************
		SNAPCAP_ERROR:
			IF NOT Enable THEN
				Internal.State := SNAPCAP_RESET;
			END_IF

	END_CASE

	Internal.FB.AsmGetShuttle();
	IF NumShuttlesFound <> 0 THEN
		FOR Internal.Index:=0 TO (NumShuttlesFound-1) DO
			Internal.FB.ShReadSegmentInfo[Internal.Index]();
			Internal.FB.ShReadInfo[Internal.Index]();
			Internal.FB.ShCopyUserData[Internal.Index]();
		END_FOR
	END_IF
	Internal.FB.GetTime();
	Internal.FB.RecipeXML();
	Internal.FB.RecipeRegPar();
	Internal.FB.DTRecipeConverter();

END_FUNCTION_BLOCK
```

#### TrakSnapSpawn.st - StarSync Implementation
```iecst
(*********************************************************************************
 * Copyright: B&R Industrial Automation GmbH
 * Author:    nealj
 * Created:   October 27, 2021/1:47 PM
 * The SnapshotSpawner FUB will gather the list of shuttles and monitor their
 * postions when enabled. When execute is TRUE, the FUB will gather the user data
 * and shuttle info of each shuttle.
 *********************************************************************************)

FUNCTION_BLOCK TrakSnapSpawn

	Internal.FB.ShCopyUserData.Mode  := mcACPTRAK_USERDATA_SET;

	Internal.FB.RecipeXML.Enable     := Enable;
	Internal.FB.RecipeXML.MpLink     := ADR(RecipeLink);
	Internal.FB.RecipeXML.DeviceName := ADR('SnapshotDevice');
	Internal.FB.RecipeXML.FileName   := ADR(SnapshotToLoad);

	Internal.FB.RecipeRegPar.Enable := Internal.FB.RecipeXML.Active;
	Internal.FB.RecipeRegPar.MpLink := ADR(RecipeLink);
	Internal.FB.RecipeRegPar.PVName := ADR(TrakSnapStructureName);

	CASE Internal.State OF
		//************************************************************************************************************
		SNAPSPAWN_IDLE:
			IF (Internal.FB.RecipeXML.Error OR Internal.FB.RecipeRegPar.Error) THEN
				//RECIPE INIT FAILED
				Error          := TRUE;
				ErrorID        := SPAWN_RECIPE_INIT_FAILED;
				Internal.State := SNAPSPAWN_ERROR;
			ELSIF (Enable AND Internal.FB.RecipeXML.Active AND Internal.FB.RecipeRegPar.Active) THEN
				Active         := TRUE;
				Ready          := TRUE;
				Internal.State := SNAPSPAWN_READY;
			END_IF

			//************************************************************************************************************
		SNAPSPAWN_READY:
			//TO DO: ADD LOGIC TO PREVENT SPAWNING SHUTTLES WITH SHUTTLES ON THE TRAK VIA ASMGETSHUTTLE FUB <~~~~~~~~~~~~~~~~~~~~~~~~~~~~~~~~~~~~~~~~~<<<
			IF NOT Enable THEN
				Internal.State := SNAPSPAWN_RESET;
			ELSIF Spawn THEN
				IF (0 = brsstrcmp(ADR(SnapshotToLoad),ADR(''))) THEN
					//SNAPSHOT TO LOAD EMPTY
					Error          := TRUE;
					ErrorID        := SPAWN_SNAPSHOT_TO_LOAD_EMPTY;
					Internal.State := SNAPSPAWN_ERROR;
				ELSE
					Done                       := FALSE;
					Ready                      := FALSE;
					Busy                       := TRUE;
					Internal.FB.RecipeXML.Load := TRUE;
					Internal.State             := SNAPSPAWN_LOAD_RECIPE;
				END_IF
			END_IF

			//************************************************************************************************************
		SNAPSPAWN_LOAD_RECIPE:
			IF NOT Enable THEN
				Internal.State := SNAPSPAWN_RESET;
			ELSIF Internal.FB.RecipeXML.Error THEN
				//LOAD RECIPE FAILED
				Error          := TRUE;
				ErrorID        := SPAWN_LOAD_RECIPE_FAILED;
				Internal.State := SNAPSPAWN_ERROR;
			ELSIF Internal.FB.RecipeXML.CommandDone THEN
				Internal.FB.RecipeXML.Load         := FALSE;
				Internal.Index                     := 0;
				IF (0 <> brsstrcmp(ADR(TrakSnapStructure.ShuttleInfo[Internal.Index].CurrentSector),ADR(''))) THEN
					//If the shuttle was on a user defined sector (the sector name is not empty), spawn it on that sector
					Internal.PV_XGETADR_ERROR_ID := PV_xgetadr(ADR(TrakSnapStructure.ShuttleInfo[Internal.Index].CurrentSector),ADR(Internal.SectorReference),ADR(Internal.SectorReferenceSize));
					Internal.FB.SecAddShuttle.Sector   := Internal.SectorReference;
					Internal.FB.SecAddShuttle.Position := TrakSnapStructure.ShuttleInfo[Internal.Index].CurrentPosition;
					Internal.FB.SecAddShuttle.Execute  := TRUE;
					Internal.State                     := SNAPSPAWN_SPAWN_SHUTTLE;
				ELSIF ((0 <> brsstrcmp(ADR(TrakSnapStructure.SegmentInfo[Internal.Index].CurrentSegment[0]),ADR('')))  OR
					   (0 <> brsstrcmp(ADR(TrakSnapStructure.SegmentInfo[Internal.Index].CurrentSegment[1]),ADR('')))  OR
					   (0 <> brsstrcmp(ADR(TrakSnapStructure.SegmentInfo[Internal.Index].CurrentSegment[2]),ADR('')))  OR
					   (0 <> brsstrcmp(ADR(TrakSnapStructure.SegmentInfo[Internal.Index].CurrentSegment[3]),ADR('')))) THEN
					//The shuttle was not on a user defined sector, and at least one of the segment references wasn't empty
					Internal.State := SNAPSPAWN_PICK_SEGSEC;
				ELSE
					//NO POSITION FOR SHUTTLE SPAWN
					Error          := TRUE;
					ErrorID        := SPAWN_NO_POS_FOR_SHUTTLE_SPAWN + Internal.Index;
				END_IF
			END_IF

			//************************************************************************************************************
		SNAPSPAWN_PICK_SEGSEC:
			//Check to see which options are valid (name is not empty and position is positive)
			Internal.SegmentSector.Valid[0] := ((0 <> brsstrcmp(ADR(TrakSnapStructure.SegmentInfo[Internal.Index].CurrentSegment[0]),ADR(''))) AND (TrakSnapStructure.SegmentInfo[Internal.Index].CurrentPosition[0] >= 0));
			Internal.SegmentSector.Valid[1] := ((0 <> brsstrcmp(ADR(TrakSnapStructure.SegmentInfo[Internal.Index].CurrentSegment[1]),ADR(''))) AND (TrakSnapStructure.SegmentInfo[Internal.Index].CurrentPosition[1] >= 0));
			Internal.SegmentSector.Valid[2] := ((0 <> brsstrcmp(ADR(TrakSnapStructure.SegmentInfo[Internal.Index].CurrentSegment[2]),ADR(''))) AND (TrakSnapStructure.SegmentInfo[Internal.Index].CurrentPosition[2] >= 0));
			Internal.SegmentSector.Valid[3] := ((0 <> brsstrcmp(ADR(TrakSnapStructure.SegmentInfo[Internal.Index].CurrentSegment[3]),ADR(''))) AND (TrakSnapStructure.SegmentInfo[Internal.Index].CurrentPosition[3] >= 0));

			//Read in the positions to improve programming readability
			Internal.SegmentSector.Position[0] := TrakSnapStructure.SegmentInfo[Internal.Index].CurrentPosition[0];
			Internal.SegmentSector.Position[1] := TrakSnapStructure.SegmentInfo[Internal.Index].CurrentPosition[1];
			Internal.SegmentSector.Position[2] := TrakSnapStructure.SegmentInfo[Internal.Index].CurrentPosition[2];
			Internal.SegmentSector.Position[3] := TrakSnapStructure.SegmentInfo[Internal.Index].CurrentPosition[3];

			//Use the for loop to determine the lowest valid segment sector position
			//This check is necessary since shuttles hanging off the end of a segment will have positions larger than the length of the segment
			FOR Internal.SegmentSector.Index:=0 TO 3 DO
				//Confirm that the best option is a valid reference
				IF Internal.SegmentSector.Valid[Internal.SegmentSector.BestOption] THEN
					//Confirm that the current index is a valid reference
					IF Internal.SegmentSector.Valid[Internal.SegmentSector.Index] THEN
						//Check if the current index is lower than the best option
						IF (Internal.SegmentSector.Position[Internal.SegmentSector.Index] < Internal.SegmentSector.Position[Internal.SegmentSector.BestOption]) THEN
							//The current index is lower than the best option, so make it the new best option
							Internal.SegmentSector.BestOption := Internal.SegmentSector.Index;
						ELSE
							//The best option is lower than the current index, so keep the best option
						END_IF
					ELSE
						//The current index is not a valid reference, so keep the best option
					END_IF
				ELSE
					//The best option is not a valid index, so make the current index the new best option
					Internal.SegmentSector.BestOption := Internal.SegmentSector.Index;
				END_IF
			END_FOR

			Internal.SectorReferenceSize       := SIZEOF(Internal.SectorReference);
			Internal.SegmentSector.Name        := '';
			brsstrcat(ADR(Internal.SegmentSector.Name),ADR(Internal.SegmentSector.Prefix));
			brsstrcat(ADR(Internal.SegmentSector.Name),ADR(TrakSnapStructure.SegmentInfo[Internal.Index].CurrentSegment[Internal.SegmentSector.BestOption]));
			Internal.PV_XGETADR_ERROR_ID       := PV_xgetadr(ADR(Internal.SegmentSector.Name),ADR(Internal.SectorReference),ADR(Internal.SectorReferenceSize));
			Internal.FB.SecAddShuttle.Sector   := Internal.SectorReference;
			Internal.FB.SecAddShuttle.Position := TrakSnapStructure.SegmentInfo[Internal.Index].CurrentPosition[Internal.SegmentSector.BestOption];
			Internal.FB.SecAddShuttle.Execute  := TRUE;
			Internal.State                     := SNAPSPAWN_SPAWN_SHUTTLE;

			//************************************************************************************************************
		SNAPSPAWN_SPAWN_SHUTTLE:
			IF NOT Enable THEN
				Internal.State := SNAPSPAWN_RESET;
			ELSIF Internal.FB.SecAddShuttle.Error THEN
				//ADD SHUTTLE FAILED
				Error          := TRUE;
				ErrorID        := SPAWN_ADD_SHUTTLE_FAILED + Internal.Index;
				Internal.State := SNAPSPAWN_ERROR;
			ELSIF Internal.FB.SecAddShuttle.Done THEN
				Internal.Shuttles[Internal.Index]      := Internal.FB.SecAddShuttle.Axis;
				Internal.FB.ShCopyUserData.Axis        := ADR(Internal.Shuttles[Internal.Index]);
				Internal.FB.SecAddShuttle.Execute      := FALSE;
				Internal.FB.ShCopyUserData.DataAddress := ADR(TrakSnapStructure.UserData[Internal.Index]);
				Internal.FB.ShCopyUserData.DataSize    := SIZEOF(TrakSnapStructure.UserData[Internal.Index]);
				Internal.FB.ShCopyUserData.Execute     := TRUE;
				Internal.State                         := SNAPSPAWN_SET_USERDATA;
			END_IF

			//************************************************************************************************************
		SNAPSPAWN_SET_USERDATA:
			IF NOT Enable THEN
				Internal.State := SNAPSPAWN_RESET;
			ELSIF Internal.FB.ShCopyUserData.Error THEN
				//SET USERDATA FAILED
				Error          := TRUE;
				ErrorID        := SPAWN_SET_USERDATA_FAILED + Internal.Index;
				Internal.State := SNAPSPAWN_ERROR;
			ELSIF Internal.FB.ShCopyUserData.Done THEN
				Internal.FB.ShCopyUserData.Execute := FALSE;
				//Check if there are more shuttles to spawn and move on
				IF (Internal.Index = (NumShuttles - 1)) THEN
					Done           := TRUE;
					Internal.State := SNAPSPAWN_DONE;
				ELSE
					Internal.Index                     := Internal.Index + 1;
					Internal.SectorReferenceSize       := SIZEOF(Internal.SectorReference);
					IF (0 <> brsstrcmp(ADR(TrakSnapStructure.ShuttleInfo[Internal.Index].CurrentSector),ADR(''))) THEN
						//If the shuttle was on a user defined sector (the sector name is not empty), spawn it on that sector
						Internal.PV_XGETADR_ERROR_ID := PV_xgetadr(ADR(TrakSnapStructure.ShuttleInfo[Internal.Index].CurrentSector),ADR(Internal.SectorReference),ADR(Internal.SectorReferenceSize));
						Internal.FB.SecAddShuttle.Sector   := Internal.SectorReference;
						Internal.FB.SecAddShuttle.Position := TrakSnapStructure.ShuttleInfo[Internal.Index].CurrentPosition;
						Internal.FB.SecAddShuttle.Execute  := TRUE;
						Internal.State                     := SNAPSPAWN_SPAWN_SHUTTLE;
					ELSIF ((0 <> brsstrcmp(ADR(TrakSnapStructure.SegmentInfo[Internal.Index].CurrentSegment[0]),ADR('')))  OR
						   (0 <> brsstrcmp(ADR(TrakSnapStructure.SegmentInfo[Internal.Index].CurrentSegment[1]),ADR('')))  OR
						   (0 <> brsstrcmp(ADR(TrakSnapStructure.SegmentInfo[Internal.Index].CurrentSegment[2]),ADR('')))  OR
						   (0 <> brsstrcmp(ADR(TrakSnapStructure.SegmentInfo[Internal.Index].CurrentSegment[3]),ADR('')))) THEN
						//The shuttle was not on a user defined sector, and at least one of the segment references wasn't empty
						Internal.State := SNAPSPAWN_PICK_SEGSEC;
					ELSE
						//NO POSITION FOR SHUTTLE SPAWN
						Error          := TRUE;
						ErrorID        := SPAWN_NO_POS_FOR_SHUTTLE_SPAWN + Internal.Index;
					END_IF
				END_IF
			END_IF

			//************************************************************************************************************
		SNAPSPAWN_DONE:
			IF NOT Enable THEN
				Internal.State := SNAPSPAWN_RESET;
			ELSIF NOT Spawn THEN
				Done           := FALSE;
				Ready          := TRUE;
				Internal.State := SNAPSPAWN_READY;
			END_IF

			//************************************************************************************************************
		SNAPSPAWN_RESET:
			Active                             := FALSE;
			Ready                              := FALSE;
			Spawn                              := FALSE;
			Busy                               := FALSE;
			Done                               := FALSE;
			Internal.FB.RecipeRegPar.Enable    := FALSE;
			Internal.FB.RecipeXML.Enable       := FALSE;
			Internal.FB.SecAddShuttle.Execute  := FALSE;
			Internal.FB.ShCopyUserData.Execute := FALSE;
			Internal.State := SNAPSPAWN_IDLE;

			//************************************************************************************************************
		SNAPSPAWN_ERROR:
			IF NOT Enable THEN
				Internal.State := SNAPSPAWN_RESET;
			END_IF

	END_CASE

	Internal.FB.RecipeRegPar();
	Internal.FB.RecipeXML();
	Internal.FB.SecAddShuttle();
	Internal.FB.ShCopyUserData();

END_FUNCTION_BLOCK
```

#### EpochConverter.st
```iecst
(*********************************************************************************
 * Copyright: B&R Industrial Automation GmbH
 * Author:    nealj
 * Created:   October 26, 2021/2:34 PM
 * Converts epoch time to a string of a format similar to DATE_AND_TIME but without
 * the ":" character. This is necessary for the recipe system. The desired format
 * is "YYYY_MM_DD HH_MM_SS".
 *********************************************************************************)

(* Converts a UDINT to a string of a format similar to DATE_AND_TIME but without the ":" character *)
FUNCTION_BLOCK EpochConverter
	CASE InternalState OF
		0:
			//Read the total number of seconds into the remainder variable
			//The offset is necessary because the calculation is off by 6hr 48min 34sec for an unknown reason
			IF (Offset = 0) THEN
				Offset := -24144;
			END_IF
			Remainder := Input + Offset;

			IF Execute THEN
				InternalState := 1;
			END_IF

		1:
			//1 year (365.24 days) = 31556926 seconds
			Year      := REAL_TO_UDINT(brmfloor((UDINT_TO_REAL(Remainder) / 31556926)));
			Remainder := Remainder - (Year   * 31556926);

			//1 month (30.44 days) = 2629743 seconds
			Month     := REAL_TO_UDINT(brmfloor((UDINT_TO_REAL(Remainder) / 2629743 )));
			Remainder := Remainder - (Month  * 2629743 );

			//1 day = 86400 seconds
			Day       := REAL_TO_UDINT(brmfloor((UDINT_TO_REAL(Remainder) / 86400   )));
			Remainder := Remainder - (Day    * 86400   );

			//1 hour = 3600 seconds
			Hour      := REAL_TO_UDINT(brmfloor((UDINT_TO_REAL(Remainder) / 3600    )));
			Remainder := Remainder - (Hour   * 3600    );

			//1 minute = 60 seconds
			Minute    := REAL_TO_UDINT(brmfloor((UDINT_TO_REAL(Remainder) / 60      )));
			Remainder := Remainder - (Minute * 60      );

			//Remainder is now the remaining seconds
			Second    := Remainder;

			//Now it must be factored in that these times represent the time since January 1, 1970 at 00:00
			Year  := Year  + 1970;
			Month := Month + 1;
			Day   := Day   + 1;

			InternalState := 2;

		2:
			//Clear the string
			brsmemset(ADR(DTString_For_Recipe),0,SIZEOF(DTString_For_Recipe));

			//Write "date"
			brsstrcat(ADR(DTString_For_Recipe),ADR(DateWord));
			brsstrcat(ADR(DTString_For_Recipe),ADR(UnderscoreCharacter));

			//Read in the year
			Year_Str := UDINT_TO_STRING(Year);
			brsstrcat(ADR(DTString_For_Recipe),ADR(Year_Str));
			brsstrcat(ADR(DTString_For_Recipe),ADR(UnderscoreCharacter));

			//Read in the month
			Month_Str := UDINT_TO_STRING(Month);
			brsstrcat(ADR(DTString_For_Recipe),ADR(Month_Str));
			brsstrcat(ADR(DTString_For_Recipe),ADR(UnderscoreCharacter));

			//Read in the day
			Day_Str := UDINT_TO_STRING(Day);
			brsstrcat(ADR(DTString_For_Recipe),ADR(Day_Str));
			brsstrcat(ADR(DTString_For_Recipe),ADR(SpaceCharacter));

			//Write "time"
			brsstrcat(ADR(DTString_For_Recipe),ADR(TimeWord));
			brsstrcat(ADR(DTString_For_Recipe),ADR(UnderscoreCharacter));

			//Read in the hour
			Hour_Str := UDINT_TO_STRING(Hour);
			brsstrcat(ADR(DTString_For_Recipe),ADR(Hour_Str));
			brsstrcat(ADR(DTString_For_Recipe),ADR(UnderscoreCharacter));

			//Read in the minute
			Minute_Str := UDINT_TO_STRING(Minute);
			brsstrcat(ADR(DTString_For_Recipe),ADR(Minute_Str));
			brsstrcat(ADR(DTString_For_Recipe),ADR(UnderscoreCharacter));

			//Read in the second
			Second_Str := UDINT_TO_STRING(Second);
			brsstrcat(ADR(DTString_For_Recipe),ADR(Second_Str));

			Execute       := FALSE;
			InternalState := 0;

	END_CASE

END_FUNCTION_BLOCK
```

### Program Logical/UserProgram (IEC)

#### Variables.var
```iecst
VAR
	AsmPowerOn : MC_BR_AsmPowerOn_AcpTrak;
	SecAddShuttle : MC_BR_SecAddShuttle_AcpTrak;
	ElasticMoveVel : MC_BR_ElasticMoveVel_AcpTrak;
	ShuttleAxis : McAxisType;
	DEV_SnapshotTaker : TrakSnapCap;
	DEV_SnapshotSpawner : TrakSnapSpawn;
	State : USINT;
	i : USINT;
END_VAR
```

#### Main.st
```iecst
(*********************************************************************************
 * Copyright: B&R Industrial Automation GmbH
 * Author:    nealj
 * Created:   November 17, 2021/3:18 PM
 *********************************************************************************)

PROGRAM _INIT
	(* Insert code here *)

END_PROGRAM

PROGRAM _CYCLIC

	DEV_SnapshotTaker.Assembly              := ADR(gAssembly_1);
	DEV_SnapshotTaker.TrakSnapStructure     := ADR(gDEV_SnapshotStructure);
	DEV_SnapshotTaker.TrakSnapStructureName := 'gDEV_SnapshotStructure';
	DEV_SnapshotTaker.RecipeLink            := ADR(gRecipeXml);
	DEV_SnapshotTaker();

	DEV_SnapshotSpawner.TrakSnapStructure     := ADR(gDEV_SnapshotStructure);
	DEV_SnapshotSpawner.TrakSnapStructureName := 'gDEV_SnapshotStructure';
	DEV_SnapshotSpawner.RecipeLink            := ADR(gRecipeXml);
	DEV_SnapshotSpawner();

END_PROGRAM

PROGRAM _EXIT
	(* Insert code here *)

END_PROGRAM
```

### Program Logical/TrakProgram (IEC)
